LIN {X -0.197,Y -544.283,Z 869.058,A 0.000,B 0.000,C 90.000,E1 46.458} C_DIS
LIN {X -0.178,Y -541.892,Z 869.055,A 0.000,B 0.000,C 90.000,E1 45.891} C_DIS
LIN {X 0.010,Y -538.422,Z 869.051,A 0.000,B 0.000,C 90.000,E1 45.162} C_DIS
LIN {X -0.016,Y -535.445,Z 869.048,A 0.000,B 0.000,C 90.000,E1 44.595} C_DIS
LIN {X -0.036,Y -532.256,Z 869.045,A 0.000,B 0.000,C 90.000,E1 44.028} C_DIS
LIN {X 0.058,Y -527.783,Z 869.041,A 0.000,B 0.000,C 90.000,E1 43.299} C_DIS
LIN {X -0.050,Y -524.016,Z 869.037,A 0.000,B 0.000,C 90.000,E1 42.732} C_DIS
LIN {X -0.151,Y -519.980,Z 869.034,A 0.000,B 0.000,C 90.000,E1 42.162} C_DIS
LIN {X 0.073,Y -515.730,Z 869.031,A 0.000,B 0.000,C 90.000,E1 41.553} C_DIS
LIN {X -0.182,Y -512.399,Z 869.029,A 0.000,B 0.000,C 90.000,E1 41.148} C_DIS
LIN {X -0.002,Y -503.778,Z 869.023,A 0.000,B 0.000,C 90.000,E1 40.092} C_DIS
LIN {X 0.166,Y -498.386,Z 869.020,A 0.000,B 0.000,C 90.000,E1 39.483} C_DIS
LIN {X -0.295,Y -491.480,Z 869.016,A 0.000,B 0.000,C 90.000,E1 38.830} C_DIS
LIN {X -0.121,Y -485.726,Z 869.013,A 0.000,B 0.000,C 90.000,E1 38.257} C_DIS
LIN {X 0.040,Y -478.343,Z 869.009,A 0.000,B 0.000,C 90.000,E1 37.569} C_DIS
LIN {X 0.098,Y -467.773,Z 869.004,A 0.000,B 0.000,C 90.000,E1 36.664} C_DIS
LIN {X -0.016,Y -456.899,Z 868.999,A 0.000,B 0.000,C 90.000,E1 35.804} C_DIS
LIN {X 0.026,Y -444.305,Z 868.994,A 0.000,B 0.000,C 90.000,E1 34.818} C_DIS
LIN {X -0.079,Y -422.825,Z 868.984,A 0.000,B 0.000,C 90.000,E1 33.086} C_DIS
LIN {X -0.077,Y -409.157,Z 868.977,A 0.000,B 0.000,C 90.000,E1 31.878} C_DIS
LIN {X 0.140,Y -401.842,Z 868.973,A 0.000,B 0.000,C 90.000,E1 31.131} C_DIS
LIN {X -0.162,Y -396.543,Z 868.970,A 0.000,B 0.000,C 90.000,E1 30.541} C_DIS
LIN {X -0.062,Y -394.558,Z 868.968,A 0.000,B 0.000,C 90.000,E1 30.256} C_DIS
LIN {X -0.054,Y -393.500,Z 868.967,A 0.000,B 0.000,C 90.000,E1 30.079} C_DIS
LIN {X 0.085,Y -391.376,Z 868.965,A 0.000,B 0.000,C 90.000,E1 29.617} C_DIS
LIN {X 0.058,Y -390.008,Z 868.961,A 0.000,B 0.000,C 90.000,E1 28.999} C_DIS
LIN {X -0.092,Y -389.501,Z 868.958,A 0.000,B 0.000,C 90.000,E1 28.487} C_DIS
LIN {X 0.127,Y -389.595,Z 868.952,A 0.000,B 0.000,C 90.000,E1 27.385} C_DIS
LIN {X -0.188,Y -392.234,Z 868.931,A 0.000,B 0.000,C 90.000,E1 23.515} C_DIS
LIN {X -0.027,Y -395.272,Z 868.913,A 0.000,B 0.000,C 90.000,E1 20.301} C_DIS
LIN {X 0.136,Y -398.327,Z 868.897,A 0.000,B 0.000,C 90.000,E1 17.457} C_DIS
LIN {X -0.006,Y -400.906,Z 868.885,A 0.000,B 0.000,C 90.000,E1 15.371} C_DIS
LIN {X -0.105,Y -405.159,Z 868.868,A 0.000,B 0.000,C 90.000,E1 12.243} C_DIS
LIN {X 0.056,Y -408.867,Z 868.854,A 0.000,B 0.000,C 90.000,E1 9.792} C_DIS
LIN {X -0.142,Y -414.004,Z 868.837,A 0.000,B 0.000,C 90.000,E1 6.720} C_DIS
LIN {X 0.028,Y -417.746,Z 868.826,A 0.000,B 0.000,C 90.000,E1 4.645} C_DIS
LIN {X -0.123,Y -423.210,Z 868.811,A 0.000,B 0.000,C 90.000,E1 1.949} C_DIS
LIN {X -0.136,Y -429.645,Z 868.795,A 0.000,B 0.000,C 90.000,E1 359.141} C_DIS
LIN {X 0.105,Y -436.193,Z 868.780,A 0.000,B 0.000,C 90.000,E1 356.445} C_DIS
LIN {X 0.117,Y -439.553,Z 868.773,A 0.000,B 0.000,C 90.000,E1 355.122} C_DIS
LIN {X -0.022,Y -442.286,Z 868.768,A 0.000,B 0.000,C 90.000,E1 354.318} C_DIS
LIN {X 0.133,Y -443.631,Z 868.767,A 0.000,B 0.000,C 90.000,E1 353.970} C_DIS
LIN {X 0.004,Y -445.225,Z 868.765,A 0.000,B 0.000,C 90.000,E1 353.685} C_DIS
LIN {X -0.182,Y -446.287,Z 868.764,A 0.000,B 0.000,C 90.000,E1 353.571} C_DIS
LIN {X 0.011,Y -448.820,Z 868.763,A 0.000,B 0.000,C 90.000,E1 353.280} C_DIS
LIN {X 0.203,Y -450.563,Z 868.762,A 0.000,B 0.000,C 90.000,E1 353.109} C_DIS
LIN {X -0.101,Y -457.050,Z 868.760,A 0.000,B 0.000,C 90.000,E1 352.761} C_DIS
LIN {X 0.066,Y -466.908,Z 868.757,A 0.000,B 0.000,C 90.000,E1 352.299} C_DIS
LIN {X -0.142,Y -476.793,Z 868.755,A 0.000,B 0.000,C 90.000,E1 351.837} C_DIS
LIN {X 0.080,Y -484.903,Z 868.752,A 0.000,B 0.000,C 90.000,E1 351.376} C_DIS
LIN {X -0.128,Y -491.410,Z 868.750,A 0.000,B 0.000,C 90.000,E1 351.027} C_DIS
LIN {X 0.259,Y -499.429,Z 868.747,A 0.000,B 0.000,C 90.000,E1 350.500} C_DIS
LIN {X 0.071,Y -510.569,Z 868.743,A 0.000,B 0.000,C 90.000,E1 349.803} C_DIS
LIN {X 0.001,Y -518.351,Z 868.741,A 0.000,B 0.000,C 90.000,E1 349.285} C_DIS
LIN {X -0.143,Y -525.997,Z 868.737,A 0.000,B 0.000,C 90.000,E1 348.757} C_DIS
LIN {X 0.082,Y -531.968,Z 868.735,A 0.000,B 0.000,C 90.000,E1 348.285} C_DIS
LIN {X 0.031,Y -540.629,Z 868.731,A 0.000,B 0.000,C 90.000,E1 347.589} C_DIS
LIN {X 0.017,Y -544.852,Z 868.729,A 0.000,B 0.000,C 90.000,E1 347.229} C_DIS
LIN {X 0.273,Y -550.376,Z 868.726,A 0.000,B 0.000,C 90.000,E1 346.700} C_DIS
LIN {X 0.133,Y -558.287,Z 868.722,A 0.000,B 0.000,C 90.000,E1 345.936} C_DIS
LIN {X -0.219,Y -562.102,Z 868.720,A 0.000,B 0.000,C 90.000,E1 345.574} C_DIS
LIN {X 0.194,Y -567.029,Z 868.717,A 0.000,B 0.000,C 90.000,E1 344.991} C_DIS
LIN {X 0.145,Y -571.768,Z 868.714,A 0.000,B 0.000,C 90.000,E1 344.448} C_DIS
LIN {X 0.065,Y -579.478,Z 868.708,A 0.000,B 0.000,C 90.000,E1 343.504} C_DIS
LIN {X 0.015,Y -584.516,Z 868.705,A 0.000,B 0.000,C 90.000,E1 342.834} C_DIS
LIN {X -0.166,Y -589.155,Z 868.701,A 0.000,B 0.000,C 90.000,E1 342.181} C_DIS
LIN {X 0.125,Y -595.226,Z 868.696,A 0.000,B 0.000,C 90.000,E1 341.221} C_DIS
LIN {X -0.081,Y -600.727,Z 868.691,A 0.000,B 0.000,C 90.000,E1 340.315} C_DIS
LIN {X -0.086,Y -607.372,Z 868.684,A 0.000,B 0.000,C 90.000,E1 339.135} C_DIS
LIN {X 0.329,Y -615.013,Z 868.676,A 0.000,B 0.000,C 90.000,E1 337.667} C_DIS
LIN {X 0.004,Y -619.578,Z 868.671,A 0.000,B 0.000,C 90.000,E1 336.794} C_DIS
LIN {X -0.271,Y -622.717,Z 868.668,A 0.000,B 0.000,C 90.000,E1 336.177} C_DIS
LIN {X 0.305,Y -626.226,Z 868.663,A 0.000,B 0.000,C 90.000,E1 335.357} C_DIS
LIN {X 0.350,Y -629.645,Z 868.659,A 0.000,B 0.000,C 90.000,E1 334.588} C_DIS
LIN {X -0.342,Y -634.773,Z 868.652,A 0.000,B 0.000,C 90.000,E1 333.384} C_DIS
LIN {X -0.161,Y -638.648,Z 868.646,A 0.000,B 0.000,C 90.000,E1 332.359} C_DIS
LIN {X 0.374,Y -642.199,Z 868.641,A 0.000,B 0.000,C 90.000,E1 331.307} C_DIS
LIN {X 0.087,Y -645.573,Z 868.635,A 0.000,B 0.000,C 90.000,E1 330.333} C_DIS
LIN {X 0.161,Y -648.796,Z 868.630,A 0.000,B 0.000,C 90.000,E1 329.331} C_DIS
LIN {X -0.185,Y -652.505,Z 868.623,A 0.000,B 0.000,C 90.000,E1 328.122} C_DIS
LIN {X -0.114,Y -654.551,Z 868.619,A 0.000,B 0.000,C 90.000,E1 327.375} C_DIS
LIN {X 0.069,Y -657.145,Z 868.613,A 0.000,B 0.000,C 90.000,E1 326.373} C_DIS
LIN {X -0.342,Y -659.954,Z 868.606,A 0.000,B 0.000,C 90.000,E1 325.182} C_DIS
LIN {X 0.218,Y -662.343,Z 868.600,A 0.000,B 0.000,C 90.000,E1 323.909} C_DIS
LIN {X -0.208,Y -664.036,Z 868.594,A 0.000,B 0.000,C 90.000,E1 322.970} C_DIS
LIN {X -0.110,Y -665.856,Z 868.587,A 0.000,B 0.000,C 90.000,E1 321.743} C_DIS
LIN {X 0.008,Y -667.448,Z 868.581,A 0.000,B 0.000,C 90.000,E1 320.517} C_DIS
LIN {X 0.061,Y -668.583,Z 868.575,A 0.000,B 0.000,C 90.000,E1 319.542} C_DIS
LIN {X 0.128,Y -669.707,Z 868.570,A 0.000,B 0.000,C 90.000,E1 318.566} C_DIS
LIN {X 0.260,Y -672.002,Z 868.558,A 0.000,B 0.000,C 90.000,E1 316.377} C_DIS
LIN {X 0.357,Y -673.553,Z 868.551,A 0.000,B 0.000,C 90.000,E1 315.162} C_DIS
LIN {X -0.053,Y -674.252,Z 868.547,A 0.000,B 0.000,C 90.000,E1 314.474} C_DIS
LIN {X -0.029,Y -674.367,Z 868.546,A 0.000,B 0.000,C 90.000,E1 314.231} C_DIS
LIN {X 0.122,Y -675.592,Z 868.539,A 0.000,B 0.000,C 90.000,E1 313.014} C_DIS
LIN {X -0.163,Y -677.036,Z 868.531,A 0.000,B 0.000,C 90.000,E1 311.595} C_DIS
LIN {X 0.044,Y -678.135,Z 868.524,A 0.000,B 0.000,C 90.000,E1 310.378} C_DIS
LIN {X -0.143,Y -679.336,Z 868.516,A 0.000,B 0.000,C 90.000,E1 308.955} C_DIS
LIN {X 0.194,Y -680.311,Z 868.510,A 0.000,B 0.000,C 90.000,E1 307.729} C_DIS
LIN {X -0.402,Y -681.261,Z 868.503,A 0.000,B 0.000,C 90.000,E1 306.583} C_DIS
LIN {X -0.035,Y -682.140,Z 868.496,A 0.000,B 0.000,C 90.000,E1 305.358} C_DIS
LIN {X 0.124,Y -683.066,Z 868.489,A 0.000,B 0.000,C 90.000,E1 303.913} C_DIS
LIN {X -0.256,Y -684.589,Z 868.477,A 0.000,B 0.000,C 90.000,E1 301.799} C_DIS
LIN {X -0.203,Y -685.887,Z 868.467,A 0.000,B 0.000,C 90.000,E1 300.129} C_DIS
LIN {X -0.171,Y -688.321,Z 868.453,A 0.000,B 0.000,C 90.000,E1 297.513} C_DIS
LIN {X -0.325,Y -689.775,Z 868.445,A 0.000,B 0.000,C 90.000,E1 296.104} C_DIS
LIN {X -0.303,Y -690.807,Z 868.440,A 0.000,B 0.000,C 90.000,E1 295.155} C_DIS
LIN {X -0.032,Y -691.777,Z 868.433,A 0.000,B 0.000,C 90.000,E1 293.951} C_DIS
LIN {X 0.168,Y -691.864,Z 868.430,A 0.000,B 0.000,C 90.000,E1 293.462} C_DIS
LIN {X -0.230,Y -691.797,Z 868.429,A 0.000,B 0.000,C 90.000,E1 293.259} C_DIS
LIN {X -0.028,Y -691.076,Z 868.427,A 0.000,B 0.000,C 90.000,E1 292.770} C_DIS
LIN {X 0.205,Y -690.377,Z 868.425,A 0.000,B 0.000,C 90.000,E1 292.514} C_DIS
LIN {X 0.286,Y -688.409,Z 868.423,A 0.000,B 0.000,C 90.000,E1 292.153} C_DIS
LIN {X -0.129,Y -686.936,Z 868.422,A 0.000,B 0.000,C 90.000,E1 291.950} C_DIS
LIN {X -0.275,Y -685.791,Z 868.421,A 0.000,B 0.000,C 90.000,E1 291.844} C_DIS
LIN {X -0.168,Y -684.078,Z 868.421,A 0.000,B 0.000,C 90.000,E1 291.716} C_DIS
LIN {X 0.160,Y -680.344,Z 868.419,A 0.000,B 0.000,C 90.000,E1 291.482} C_DIS
LIN {X -0.041,Y -676.937,Z 868.419,A 0.000,B 0.000,C 90.000,E1 291.334} C_DIS
LIN {X -0.144,Y -670.811,Z 868.417,A 0.000,B 0.000,C 90.000,E1 291.153} C_DIS
LIN {X -0.224,Y -658.370,Z 868.416,A 0.000,B 0.000,C 90.000,E1 290.844} C_DIS
LIN {X 0.181,Y -654.807,Z 868.415,A 0.000,B 0.000,C 90.000,E1 290.684} C_DIS
LIN {X -0.260,Y -652.134,Z 868.414,A 0.000,B 0.000,C 90.000,E1 290.610} C_DIS
LIN {X -0.212,Y -650.429,Z 868.414,A 0.000,B 0.000,C 90.000,E1 290.482} C_DIS
LIN {X 0.072,Y -649.078,Z 868.413,A 0.000,B 0.000,C 90.000,E1 290.355} C_DIS
LIN {X 0.034,Y -649.065,Z 868.413,A 0.000,B 0.000,C 90.000,E1 290.355} C_DIS
LIN {X -0.066,Y -648.618,Z 868.412,A 0.000,B 0.000,C 90.000,E1 290.248} C_DIS
LIN {X -0.110,Y -648.618,Z 868.412,A 0.000,B 0.000,C 90.000,E1 290.248} C_DIS
LIN {X -0.132,Y -649.438,Z 868.410,A 0.000,B 0.000,C 90.000,E1 289.885} C_DIS
LIN {X -0.167,Y -652.192,Z 868.407,A 0.000,B 0.000,C 90.000,E1 289.268} C_DIS
LIN {X 0.241,Y -658.845,Z 868.400,A 0.000,B 0.000,C 90.000,E1 288.000} C_DIS
LIN {X 0.117,Y -662.385,Z 868.396,A 0.000,B 0.000,C 90.000,E1 287.275} C_DIS
LIN {X 0.021,Y -665.410,Z 868.392,A 0.000,B 0.000,C 90.000,E1 286.551} C_DIS
LIN {X -0.153,Y -667.161,Z 868.389,A 0.000,B 0.000,C 90.000,E1 286.079} C_DIS
LIN {X -0.389,Y -669.411,Z 868.385,A 0.000,B 0.000,C 90.000,E1 285.371} C_DIS
LIN {X 0.288,Y -670.650,Z 868.383,A 0.000,B 0.000,C 90.000,E1 284.828} C_DIS
LIN {X 0.023,Y -672.437,Z 868.377,A 0.000,B 0.000,C 90.000,E1 283.883} C_DIS
LIN {X -0.040,Y -672.850,Z 868.376,A 0.000,B 0.000,C 90.000,E1 283.647} C_DIS
LIN {X 0.377,Y -673.880,Z 868.370,A 0.000,B 0.000,C 90.000,E1 282.647} C_DIS
LIN {X 0.062,Y -674.337,Z 868.366,A 0.000,B 0.000,C 90.000,E1 281.951} C_DIS
LIN {X -0.109,Y -674.352,Z 868.362,A 0.000,B 0.000,C 90.000,E1 281.243} C_DIS
LIN {X -0.354,Y -674.152,Z 868.360,A 0.000,B 0.000,C 90.000,E1 280.782} C_DIS
LIN {X 0.189,Y -673.702,Z 868.357,A 0.000,B 0.000,C 90.000,E1 280.254} C_DIS
LIN {X -0.052,Y -672.960,Z 868.354,A 0.000,B 0.000,C 90.000,E1 279.792} C_DIS
LIN {X -0.184,Y -671.934,Z 868.352,A 0.000,B 0.000,C 90.000,E1 279.321} C_DIS
LIN {X 0.230,Y -670.570,Z 868.349,A 0.000,B 0.000,C 90.000,E1 278.803} C_DIS
LIN {X -0.024,Y -668.909,Z 868.346,A 0.000,B 0.000,C 90.000,E1 278.341} C_DIS
LIN {X -0.107,Y -668.021,Z 868.345,A 0.000,B 0.000,C 90.000,E1 278.106} C_DIS
LIN {X 0.286,Y -665.917,Z 868.342,A 0.000,B 0.000,C 90.000,E1 277.587} C_DIS
LIN {X -0.006,Y -662.895,Z 868.339,A 0.000,B 0.000,C 90.000,E1 277.004} C_DIS
LIN {X 0.346,Y -660.140,Z 868.336,A 0.000,B 0.000,C 90.000,E1 276.486} C_DIS
LIN {X -0.077,Y -656.035,Z 868.333,A 0.000,B 0.000,C 90.000,E1 275.910} C_DIS
LIN {X 0.227,Y -652.239,Z 868.330,A 0.000,B 0.000,C 90.000,E1 275.391} C_DIS
LIN {X -0.258,Y -646.569,Z 868.327,A 0.000,B 0.000,C 90.000,E1 274.816} C_DIS
LIN {X 0.058,Y -641.662,Z 868.324,A 0.000,B 0.000,C 90.000,E1 274.302} C_DIS
LIN {X -0.051,Y -636.315,Z 868.321,A 0.000,B 0.000,C 90.000,E1 273.841} C_DIS
LIN {X 0.009,Y -630.719,Z 868.319,A 0.000,B 0.000,C 90.000,E1 273.383} C_DIS
LIN {X -0.187,Y -624.915,Z 868.317,A 0.000,B 0.000,C 90.000,E1 272.980} C_DIS
LIN {X 0.116,Y -617.299,Z 868.314,A 0.000,B 0.000,C 90.000,E1 272.465} C_DIS
LIN {X -0.126,Y -610.630,Z 868.312,A 0.000,B 0.000,C 90.000,E1 272.121} C_DIS
LIN {X -0.022,Y -603.828,Z 868.310,A 0.000,B 0.000,C 90.000,E1 271.776} C_DIS
LIN {X -0.152,Y -596.472,Z 868.308,A 0.000,B 0.000,C 90.000,E1 271.489} C_DIS
LIN {X 0.194,Y -591.084,Z 868.307,A 0.000,B 0.000,C 90.000,E1 271.260} C_DIS
LIN {X 0.273,Y -583.480,Z 868.306,A 0.000,B 0.000,C 90.000,E1 271.031} C_DIS
LIN {X 0.109,Y -577.567,Z 868.305,A 0.000,B 0.000,C 90.000,E1 270.917} C_DIS
LIN {X 0.132,Y -571.301,Z 868.305,A 0.000,B 0.000,C 90.000,E1 270.802} C_DIS
LIN {X -0.095,Y -564.097,Z 868.304,A 0.000,B 0.000,C 90.000,E1 270.745} C_DIS
LIN {X -0.109,Y -552.668,Z 868.304,A 0.000,B 0.000,C 90.000,E1 270.688} C_DIS
LIN {X 0.187,Y -549.596,Z 868.303,A 0.000,B 0.000,C 90.000,E1 270.573} C_DIS
LIN {X 0.157,Y -549.518,Z 868.303,A 0.000,B 0.000,C 90.000,E1 270.573} C_DIS
LIN {X -0.177,Y -547.454,Z 868.302,A 0.000,B 0.000,C 90.000,E1 270.344} C_DIS
LIN {X 0.153,Y -546.964,Z 868.301,A 0.000,B 0.000,C 90.000,E1 270.172} C_DIS
LIN {X -0.068,Y -545.980,Z 868.298,A 0.000,B 0.000,C 90.000,E1 269.714} C_DIS
LIN {X 0.180,Y -544.198,Z 868.289,A 0.000,B 0.000,C 90.000,E1 267.993} C_DIS
LIN {X -0.065,Y -542.539,Z 868.276,A 0.000,B 0.000,C 90.000,E1 265.755} C_DIS
LIN {X 0.132,Y -541.407,Z 868.267,A 0.000,B 0.000,C 90.000,E1 264.033} C_DIS
LIN {X -0.193,Y -540.299,Z 868.259,A 0.000,B 0.000,C 90.000,E1 262.648} C_DIS
LIN {X 0.143,Y -538.737,Z 868.250,A 0.000,B 0.000,C 90.000,E1 260.905} C_DIS
LIN {X -0.077,Y -537.063,Z 868.240,A 0.000,B 0.000,C 90.000,E1 259.218} C_DIS
LIN {X 0.172,Y -535.823,Z 868.234,A 0.000,B 0.000,C 90.000,E1 258.049} C_DIS
LIN {X -0.123,Y -534.523,Z 868.227,A 0.000,B 0.000,C 90.000,E1 256.937} C_DIS
LIN {X 0.247,Y -532.762,Z 868.219,A 0.000,B 0.000,C 90.000,E1 255.463} C_DIS
LIN {X 0.062,Y -531.010,Z 868.211,A 0.000,B 0.000,C 90.000,E1 254.047} C_DIS
LIN {X 0.159,Y -528.989,Z 868.202,A 0.000,B 0.000,C 90.000,E1 252.308} C_DIS
LIN {X 0.200,Y -527.579,Z 868.195,A 0.000,B 0.000,C 90.000,E1 251.148} C_DIS
LIN {X 0.221,Y -525.670,Z 868.187,A 0.000,B 0.000,C 90.000,E1 249.699} C_DIS
LIN {X -0.106,Y -523.660,Z 868.179,A 0.000,B 0.000,C 90.000,E1 248.284} C_DIS
LIN {X 0.212,Y -521.516,Z 868.171,A 0.000,B 0.000,C 90.000,E1 246.794} C_DIS
LIN {X -0.135,Y -519.738,Z 868.165,A 0.000,B 0.000,C 90.000,E1 245.665} C_DIS
LIN {X -0.018,Y -517.017,Z 868.155,A 0.000,B 0.000,C 90.000,E1 243.896} C_DIS
LIN {X -0.196,Y -514.052,Z 868.145,A 0.000,B 0.000,C 90.000,E1 242.153} C_DIS
LIN {X -0.106,Y -510.431,Z 868.134,A 0.000,B 0.000,C 90.000,E1 240.078} C_DIS
LIN {X 0.099,Y -508.251,Z 868.127,A 0.000,B 0.000,C 90.000,E1 238.869} C_DIS
LIN {X -0.155,Y -506.003,Z 868.121,A 0.000,B 0.000,C 90.000,E1 237.709} C_DIS
LIN {X -0.127,Y -503.122,Z 868.112,A 0.000,B 0.000,C 90.000,E1 236.215} C_DIS
LIN {X -0.054,Y -501.273,Z 868.107,A 0.000,B 0.000,C 90.000,E1 235.308} C_DIS
LIN {X -0.125,Y -498.475,Z 868.101,A 0.000,B 0.000,C 90.000,E1 234.116} C_DIS
LIN {X -0.077,Y -494.841,Z 868.092,A 0.000,B 0.000,C 90.000,E1 232.603} C_DIS
LIN {X -0.094,Y -489.786,Z 868.080,A 0.000,B 0.000,C 90.000,E1 230.481} C_DIS
LIN {X 0.089,Y -486.326,Z 868.072,A 0.000,B 0.000,C 90.000,E1 228.933} C_DIS
LIN {X 0.219,Y -480.908,Z 868.058,A 0.000,B 0.000,C 90.000,E1 226.458} C_DIS
LIN {X -0.063,Y -476.891,Z 868.048,A 0.000,B 0.000,C 90.000,E1 224.636} C_DIS
LIN {X -0.174,Y -475.534,Z 868.045,A 0.000,B 0.000,C 90.000,E1 224.028} C_DIS
LIN {X -0.131,Y -470.766,Z 868.032,A 0.000,B 0.000,C 90.000,E1 221.838} C_DIS
LIN {X 0.060,Y -466.660,Z 868.022,A 0.000,B 0.000,C 90.000,E1 219.930} C_DIS
LIN {X -0.041,Y -461.947,Z 868.010,A 0.000,B 0.000,C 90.000,E1 217.729} C_DIS
LIN {X -0.026,Y -458.644,Z 868.001,A 0.000,B 0.000,C 90.000,E1 216.137} C_DIS
LIN {X 0.125,Y -454.560,Z 867.990,A 0.000,B 0.000,C 90.000,E1 214.199} C_DIS
LIN {X -0.272,Y -449.041,Z 867.976,A 0.000,B 0.000,C 90.000,E1 211.671} C_DIS
LIN {X 0.107,Y -445.582,Z 867.967,A 0.000,B 0.000,C 90.000,E1 210.001} C_DIS
LIN {X 0.033,Y -441.445,Z 867.956,A 0.000,B 0.000,C 90.000,E1 208.052} C_DIS
LIN {X -0.113,Y -436.579,Z 867.943,A 0.000,B 0.000,C 90.000,E1 205.771} C_DIS
LIN {X 0.001,Y -432.360,Z 867.932,A 0.000,B 0.000,C 90.000,E1 203.770} C_DIS
LIN {X 0.048,Y -429.001,Z 867.923,A 0.000,B 0.000,C 90.000,E1 202.099} C_DIS
LIN {X 0.029,Y -425.565,Z 867.914,A 0.000,B 0.000,C 90.000,E1 200.429} C_DIS
LIN {X -0.034,Y -421.585,Z 867.902,A 0.000,B 0.000,C 90.000,E1 198.417} C_DIS
LIN {X 0.137,Y -418.994,Z 867.895,A 0.000,B 0.000,C 90.000,E1 197.040} C_DIS
LIN {X -0.136,Y -416.226,Z 867.887,A 0.000,B 0.000,C 90.000,E1 195.717} C_DIS
LIN {X -0.130,Y -412.786,Z 867.878,A 0.000,B 0.000,C 90.000,E1 194.008} C_DIS
LIN {X -0.056,Y -408.051,Z 867.864,A 0.000,B 0.000,C 90.000,E1 191.591} C_DIS
LIN {X 0.013,Y -405.331,Z 867.857,A 0.000,B 0.000,C 90.000,E1 190.197} C_DIS
LIN {X 0.042,Y -401.878,Z 867.847,A 0.000,B 0.000,C 90.000,E1 188.454} C_DIS
LIN {X 0.085,Y -394.628,Z 867.826,A 0.000,B 0.000,C 90.000,E1 184.588} C_DIS
LIN {X 0.054,Y -388.590,Z 867.804,A 0.000,B 0.000,C 90.000,E1 180.688} C_DIS
LIN {X -0.022,Y -386.099,Z 867.794,A 0.000,B 0.000,C 90.000,E1 178.912} C_DIS
LIN {X -0.143,Y -383.551,Z 867.784,A 0.000,B 0.000,C 90.000,E1 177.135} C_DIS
LIN {X 0.081,Y -380.945,Z 867.774,A 0.000,B 0.000,C 90.000,E1 175.298} C_DIS
LIN {X -0.126,Y -376.593,Z 867.756,A 0.000,B 0.000,C 90.000,E1 172.064} C_DIS
LIN {X 0.117,Y -373.744,Z 867.740,A 0.000,B 0.000,C 90.000,E1 169.106} C_DIS
LIN {X -0.037,Y -373.143,Z 867.729,A 0.000,B 0.000,C 90.000,E1 167.297} C_DIS
LIN {X -0.200,Y -373.065,Z 867.725,A 0.000,B 0.000,C 90.000,E1 166.589} C_DIS
LIN {X -0.036,Y -373.482,Z 867.719,A 0.000,B 0.000,C 90.000,E1 165.463} C_DIS
LIN {X -0.198,Y -374.026,Z 867.715,A 0.000,B 0.000,C 90.000,E1 164.755} C_DIS
LIN {X 0.106,Y -375.078,Z 867.711,A 0.000,B 0.000,C 90.000,E1 163.976} C_DIS
LIN {X -0.045,Y -376.748,Z 867.707,A 0.000,B 0.000,C 90.000,E1 163.268} C_DIS
LIN {X -0.071,Y -378.591,Z 867.704,A 0.000,B 0.000,C 90.000,E1 162.725} C_DIS
LIN {X -0.084,Y -382.638,Z 867.700,A 0.000,B 0.000,C 90.000,E1 162.000} C_DIS
LIN {X 0.046,Y -388.965,Z 867.696,A 0.000,B 0.000,C 90.000,E1 161.329} C_DIS
LIN {X -0.154,Y -392.565,Z 867.695,A 0.000,B 0.000,C 90.000,E1 161.094} C_DIS
LIN {X 0.057,Y -396.273,Z 867.694,A 0.000,B 0.000,C 90.000,E1 160.859} C_DIS
LIN {X -0.075,Y -407.283,Z 867.691,A 0.000,B 0.000,C 90.000,E1 160.369} C_DIS
LIN {X 0.119,Y -412.241,Z 867.690,A 0.000,B 0.000,C 90.000,E1 160.115} C_DIS
LIN {X -0.076,Y -422.368,Z 867.687,A 0.000,B 0.000,C 90.000,E1 159.625} C_DIS
LIN {X -0.111,Y -428.851,Z 867.685,A 0.000,B 0.000,C 90.000,E1 159.263} C_DIS
LIN {X 0.158,Y -432.122,Z 867.684,A 0.000,B 0.000,C 90.000,E1 159.028} C_DIS
LIN {X 0.185,Y -438.265,Z 867.681,A 0.000,B 0.000,C 90.000,E1 158.592} C_DIS
LIN {X -0.013,Y -444.685,Z 867.679,A 0.000,B 0.000,C 90.000,E1 158.156} C_DIS
LIN {X -0.023,Y -452.335,Z 867.675,A 0.000,B 0.000,C 90.000,E1 157.539} C_DIS
LIN {X 0.079,Y -459.657,Z 867.672,A 0.000,B 0.000,C 90.000,E1 156.869} C_DIS
LIN {X -0.130,Y -464.014,Z 867.669,A 0.000,B 0.000,C 90.000,E1 156.485} C_DIS
LIN {X 0.116,Y -475.059,Z 867.663,A 0.000,B 0.000,C 90.000,E1 155.305} C_DIS
LIN {X 0.141,Y -480.397,Z 867.660,A 0.000,B 0.000,C 90.000,E1 154.717} C_DIS
LIN {X 0.080,Y -486.875,Z 867.656,A 0.000,B 0.000,C 90.000,E1 153.973} C_DIS
LIN {X 0.126,Y -492.956,Z 867.651,A 0.000,B 0.000,C 90.000,E1 153.204} C_DIS
LIN {X -0.267,Y -504.284,Z 867.643,A 0.000,B 0.000,C 90.000,E1 151.769} C_DIS
LIN {X -0.152,Y -507.524,Z 867.641,A 0.000,B 0.000,C 90.000,E1 151.307} C_DIS
LIN {X -0.031,Y -514.896,Z 867.635,A 0.000,B 0.000,C 90.000,E1 150.255} C_DIS
LIN {X 0.149,Y -517.786,Z 867.632,A 0.000,B 0.000,C 90.000,E1 149.793} C_DIS
LIN {X -0.193,Y -519.767,Z 867.631,A 0.000,B 0.000,C 90.000,E1 149.537} C_DIS
LIN {X 0.016,Y -522.734,Z 867.628,A 0.000,B 0.000,C 90.000,E1 149.076} C_DIS
LIN {X 0.035,Y -528.210,Z 867.623,A 0.000,B 0.000,C 90.000,E1 148.201} C_DIS
LIN {X 0.114,Y -533.412,Z 867.619,A 0.000,B 0.000,C 90.000,E1 147.327} C_DIS
LIN {X -0.343,Y -540.754,Z 867.611,A 0.000,B 0.000,C 90.000,E1 146.087} C_DIS
LIN {X 0.172,Y -545.299,Z 867.607,A 0.000,B 0.000,C 90.000,E1 145.182} C_DIS
LIN {X 0.218,Y -551.991,Z 867.600,A 0.000,B 0.000,C 90.000,E1 143.909} C_DIS
LIN {X 0.087,Y -556.383,Z 867.595,A 0.000,B 0.000,C 90.000,E1 143.084} C_DIS
LIN {X 0.076,Y -563.544,Z 867.587,A 0.000,B 0.000,C 90.000,E1 141.698} C_DIS
LIN {X -0.245,Y -570.774,Z 867.580,A 0.000,B 0.000,C 90.000,E1 140.356} C_DIS
LIN {X 0.011,Y -573.577,Z 867.577,A 0.000,B 0.000,C 90.000,E1 139.784} C_DIS
LIN {X -0.033,Y -579.444,Z 867.570,A 0.000,B 0.000,C 90.000,E1 138.566} C_DIS
LIN {X 0.119,Y -591.123,Z 867.556,A 0.000,B 0.000,C 90.000,E1 136.134} C_DIS
LIN {X -0.089,Y -596.837,Z 867.550,A 0.000,B 0.000,C 90.000,E1 134.960} C_DIS
LIN {X 0.018,Y -603.677,Z 867.542,A 0.000,B 0.000,C 90.000,E1 133.500} C_DIS
LIN {X -0.111,Y -609.461,Z 867.534,A 0.000,B 0.000,C 90.000,E1 132.204} C_DIS
LIN {X 0.066,Y -614.106,Z 867.529,A 0.000,B 0.000,C 90.000,E1 131.148} C_DIS
LIN {X 0.143,Y -619.325,Z 867.521,A 0.000,B 0.000,C 90.000,E1 129.850} C_DIS
LIN {X -0.096,Y -624.303,Z 867.514,A 0.000,B 0.000,C 90.000,E1 128.588} C_DIS
LIN {X -0.304,Y -626.304,Z 867.512,A 0.000,B 0.000,C 90.000,E1 128.096} C_DIS
LIN {X 0.275,Y -633.863,Z 867.500,A 0.000,B 0.000,C 90.000,E1 126.011} C_DIS
LIN {X 0.010,Y -637.284,Z 867.495,A 0.000,B 0.000,C 90.000,E1 125.025} C_DIS
LIN {X 0.316,Y -640.438,Z 867.489,A 0.000,B 0.000,C 90.000,E1 123.992} C_DIS
LIN {X -0.271,Y -642.596,Z 867.485,A 0.000,B 0.000,C 90.000,E1 123.293} C_DIS
LIN {X 0.183,Y -644.109,Z 867.482,A 0.000,B 0.000,C 90.000,E1 122.752} C_DIS
LIN {X 0.167,Y -645.929,Z 867.478,A 0.000,B 0.000,C 90.000,E1 122.005} C_DIS
LIN {X -0.243,Y -646.909,Z 867.475,A 0.000,B 0.000,C 90.000,E1 121.544} C_DIS
LIN {X 0.245,Y -648.089,Z 867.472,A 0.000,B 0.000,C 90.000,E1 121.003} C_DIS
LIN {X 0.265,Y -649.593,Z 867.468,A 0.000,B 0.000,C 90.000,E1 120.256} C_DIS
LIN {X 0.163,Y -651.642,Z 867.461,A 0.000,B 0.000,C 90.000,E1 119.027} C_DIS
LIN {X -0.209,Y -652.474,Z 867.459,A 0.000,B 0.000,C 90.000,E1 118.565} C_DIS
LIN {X 0.307,Y -653.102,Z 867.456,A 0.000,B 0.000,C 90.000,E1 118.025} C_DIS
LIN {X 0.045,Y -654.272,Z 867.452,A 0.000,B 0.000,C 90.000,E1 117.308} C_DIS
LIN {X 0.198,Y -655.731,Z 867.446,A 0.000,B 0.000,C 90.000,E1 116.309} C_DIS
LIN {X -0.159,Y -656.272,Z 867.444,A 0.000,B 0.000,C 90.000,E1 115.848} C_DIS
LIN {X 0.152,Y -657.228,Z 867.437,A 0.000,B 0.000,C 90.000,E1 114.591} C_DIS
LIN {X -0.208,Y -657.292,Z 867.434,A 0.000,B 0.000,C 90.000,E1 114.131} C_DIS
LIN {X -0.239,Y -657.057,Z 867.431,A 0.000,B 0.000,C 90.000,E1 113.643} C_DIS
LIN {X -0.122,Y -656.742,Z 867.430,A 0.000,B 0.000,C 90.000,E1 113.387} C_DIS
LIN {X -0.150,Y -654.997,Z 867.427,A 0.000,B 0.000,C 90.000,E1 112.898} C_DIS
LIN {X -0.095,Y -654.441,Z 867.427,A 0.000,B 0.000,C 90.000,E1 112.770} C_DIS
LIN {X 0.012,Y -652.332,Z 867.425,A 0.000,B 0.000,C 90.000,E1 112.514} C_DIS
LIN {X 0.043,Y -650.133,Z 867.423,A 0.000,B 0.000,C 90.000,E1 112.206} C_DIS
LIN {X 0.067,Y -645.868,Z 867.421,A 0.000,B 0.000,C 90.000,E1 111.844} C_DIS
LIN {X 0.241,Y -644.434,Z 867.421,A 0.000,B 0.000,C 90.000,E1 111.716} C_DIS
LIN {X -0.140,Y -642.738,Z 867.420,A 0.000,B 0.000,C 90.000,E1 111.642} C_DIS
LIN {X -0.001,Y -635.779,Z 867.418,A 0.000,B 0.000,C 90.000,E1 111.280} C_DIS
LIN {X 0.280,Y -624.282,Z 867.416,A 0.000,B 0.000,C 90.000,E1 110.791} C_DIS
LIN {X 0.206,Y -620.716,Z 867.415,A 0.000,B 0.000,C 90.000,E1 110.663} C_DIS
LIN {X -0.169,Y -607.291,Z 867.412,A 0.000,B 0.000,C 90.000,E1 110.120} C_DIS
LIN {X -0.087,Y -594.600,Z 867.408,A 0.000,B 0.000,C 90.000,E1 109.504} C_DIS
LIN {X -0.178,Y -588.018,Z 867.407,A 0.000,B 0.000,C 90.000,E1 109.214} C_DIS
LIN {X 0.202,Y -580.675,Z 867.405,A 0.000,B 0.000,C 90.000,E1 108.906} C_DIS
LIN {X -0.044,Y -566.311,Z 867.403,A 0.000,B 0.000,C 90.000,E1 108.489} C_DIS
LIN {X 0.127,Y -565.064,Z 867.402,A 0.000,B 0.000,C 90.000,E1 108.417} C_DIS
LIN {X 0.152,Y -562.083,Z 867.401,A 0.000,B 0.000,C 90.000,E1 108.236} C_DIS
LIN {X -0.016,Y -560.581,Z 867.400,A 0.000,B 0.000,C 90.000,E1 108.055} C_DIS
LIN {X -0.129,Y -560.028,Z 867.400,A 0.000,B 0.000,C 90.000,E1 107.928} C_DIS
LIN {X 0.002,Y -559.229,Z 867.398,A 0.000,B 0.000,C 90.000,E1 107.638} C_DIS
LIN {X -0.176,Y -558.740,Z 867.396,A 0.000,B 0.000,C 90.000,E1 107.221} C_DIS
LIN {X -0.089,Y -559.396,Z 867.377,A 0.000,B 0.000,C 90.000,E1 103.883} C_DIS
LIN {X -0.305,Y -560.228,Z 867.368,A 0.000,B 0.000,C 90.000,E1 102.243} C_DIS
LIN {X -0.196,Y -561.731,Z 867.356,A 0.000,B 0.000,C 90.000,E1 100.018} C_DIS
LIN {X 0.173,Y -562.329,Z 867.351,A 0.000,B 0.000,C 90.000,E1 99.151} C_DIS
LIN {X -0.170,Y -563.476,Z 867.342,A 0.000,B 0.000,C 90.000,E1 97.530} C_DIS
LIN {X -0.182,Y -564.140,Z 867.336,A 0.000,B 0.000,C 90.000,E1 96.429} C_DIS
LIN {X -0.009,Y -564.944,Z 867.326,A 0.000,B 0.000,C 90.000,E1 94.759} C_DIS
LIN {X 0.130,Y -565.559,Z 867.317,A 0.000,B 0.000,C 90.000,E1 93.094} C_DIS
LIN {X 0.253,Y -566.082,Z 867.308,A 0.000,B 0.000,C 90.000,E1 91.432} C_DIS
LIN {X 0.148,Y -566.358,Z 867.302,A 0.000,B 0.000,C 90.000,E1 90.344} C_DIS
LIN {X 0.166,Y -566.730,Z 867.294,A 0.000,B 0.000,C 90.000,E1 88.969} C_DIS
LIN {X -0.134,Y -567.048,Z 867.284,A 0.000,B 0.000,C 90.000,E1 87.078} C_DIS
LIN {X 0.052,Y -567.329,Z 867.275,A 0.000,B 0.000,C 90.000,E1 85.412} C_DIS
LIN {X 0.025,Y -567.532,Z 867.268,A 0.000,B 0.000,C 90.000,E1 84.318} C_DIS
LIN {X 0.172,Y -567.786,Z 867.261,A 0.000,B 0.000,C 90.000,E1 82.932} C_DIS
LIN {X 0.208,Y -568.422,Z 867.249,A 0.000,B 0.000,C 90.000,E1 80.735} C_DIS
LIN {X 0.072,Y -568.974,Z 867.240,A 0.000,B 0.000,C 90.000,E1 79.106} C_DIS
LIN {X 0.244,Y -569.824,Z 867.229,A 0.000,B 0.000,C 90.000,E1 77.173} C_DIS
LIN {X 0.055,Y -570.298,Z 867.221,A 0.000,B 0.000,C 90.000,E1 75.825} C_DIS
LIN {X -0.028,Y -570.963,Z 867.211,A 0.000,B 0.000,C 90.000,E1 73.921} C_DIS
LIN {X -0.277,Y -571.227,Z 867.202,A 0.000,B 0.000,C 90.000,E1 72.308} C_DIS
LIN {X -0.326,Y -571.340,Z 867.196,A 0.000,B 0.000,C 90.000,E1 71.221} C_DIS
LIN {X -0.205,Y -571.453,Z 867.186,A 0.000,B 0.000,C 90.000,E1 69.571} C_DIS
LIN {X -0.084,Y -571.446,Z 867.177,A 0.000,B 0.000,C 90.000,E1 67.922} C_DIS
LIN {X -0.055,Y -571.493,Z 867.168,A 0.000,B 0.000,C 90.000,E1 66.282} C_DIS
LIN {X -0.254,Y -571.332,Z 867.159,A 0.000,B 0.000,C 90.000,E1 64.665} C_DIS
LIN {X 0.190,Y -571.026,Z 867.152,A 0.000,B 0.000,C 90.000,E1 63.256} C_DIS
LIN {X 0.122,Y -570.681,Z 867.144,A 0.000,B 0.000,C 90.000,E1 61.897} C_DIS
LIN {X 0.041,Y -570.134,Z 867.136,A 0.000,B 0.000,C 90.000,E1 60.539} C_DIS
LIN {X -0.199,Y -569.799,Z 867.132,A 0.000,B 0.000,C 90.000,E1 59.744} C_DIS
LIN {X 0.086,Y -568.585,Z 867.123,A 0.000,B 0.000,C 90.000,E1 58.074} C_DIS
LIN {X 0.128,Y -567.906,Z 867.118,A 0.000,B 0.000,C 90.000,E1 57.248} C_DIS
LIN {X 0.052,Y -567.420,Z 867.115,A 0.000,B 0.000,C 90.000,E1 56.707} C_DIS
LIN {X 0.200,Y -566.147,Z 867.109,A 0.000,B 0.000,C 90.000,E1 55.595} C_DIS
LIN {X -0.130,Y -564.674,Z 867.103,A 0.000,B 0.000,C 90.000,E1 54.529} C_DIS
LIN {X -0.022,Y -563.053,Z 867.097,A 0.000,B 0.000,C 90.000,E1 53.417} C_DIS
LIN {X 0.291,Y -561.682,Z 867.092,A 0.000,B 0.000,C 90.000,E1 52.557} C_DIS
LIN {X 0.145,Y -560.141,Z 867.088,A 0.000,B 0.000,C 90.000,E1 51.743} C_DIS
LIN {X -0.013,Y -558.407,Z 867.083,A 0.000,B 0.000,C 90.000,E1 50.928} C_DIS
LIN {X 0.239,Y -556.364,Z 867.078,A 0.000,B 0.000,C 90.000,E1 50.070} C_DIS
LIN {X 0.035,Y -553.975,Z 867.074,A 0.000,B 0.000,C 90.000,E1 49.256} C_DIS
LIN {X 0.110,Y -552.288,Z 867.071,A 0.000,B 0.000,C 90.000,E1 48.690} C_DIS
LIN {X -0.139,Y -549.403,Z 867.066,A 0.000,B 0.000,C 90.000,E1 47.877} C_DIS
LIN {X -0.088,Y -547.301,Z 867.063,A 0.000,B 0.000,C 90.000,E1 47.310} C_DIS
LIN {X -0.025,Y -543.850,Z 867.058,A 0.000,B 0.000,C 90.000,E1 46.458} C_DIS
LIN {X 0.180,Y -540.691,Z 867.054,A 0.000,B 0.000,C 90.000,E1 45.729} C_DIS
LIN {X 0.170,Y -537.892,Z 867.051,A 0.000,B 0.000,C 90.000,E1 45.162} C_DIS
LIN {X 0.140,Y -534.859,Z 867.048,A 0.000,B 0.000,C 90.000,E1 44.595} C_DIS
LIN {X 0.258,Y -530.677,Z 867.044,A 0.000,B 0.000,C 90.000,E1 43.866} C_DIS
LIN {X 0.173,Y -527.060,Z 867.041,A 0.000,B 0.000,C 90.000,E1 43.299} C_DIS
LIN {X -0.095,Y -524.262,Z 867.038,A 0.000,B 0.000,C 90.000,E1 42.894} C_DIS
LIN {X 0.155,Y -520.204,Z 867.035,A 0.000,B 0.000,C 90.000,E1 42.285} C_DIS
LIN {X 0.031,Y -515.908,Z 867.032,A 0.000,B 0.000,C 90.000,E1 41.714} C_DIS
LIN {X -0.068,Y -511.397,Z 867.029,A 0.000,B 0.000,C 90.000,E1 41.148} C_DIS
LIN {X -0.014,Y -503.954,Z 867.024,A 0.000,B 0.000,C 90.000,E1 40.253} C_DIS
LIN {X 0.167,Y -498.621,Z 867.020,A 0.000,B 0.000,C 90.000,E1 39.644} C_DIS
LIN {X 0.007,Y -493.249,Z 867.017,A 0.000,B 0.000,C 90.000,E1 39.116} C_DIS
LIN {X 0.062,Y -487.932,Z 867.014,A 0.000,B 0.000,C 90.000,E1 38.588} C_DIS
LIN {X 0.011,Y -482.074,Z 867.011,A 0.000,B 0.000,C 90.000,E1 38.051} C_DIS
LIN {X 0.042,Y -477.565,Z 867.009,A 0.000,B 0.000,C 90.000,E1 37.649} C_DIS
LIN {X 0.143,Y -468.567,Z 867.005,A 0.000,B 0.000,C 90.000,E1 36.870} C_DIS
LIN {X 0.062,Y -456.101,Z 866.999,A 0.000,B 0.000,C 90.000,E1 35.884} C_DIS
LIN {X -0.195,Y -441.953,Z 866.993,A 0.000,B 0.000,C 90.000,E1 34.818} C_DIS
LIN {X 0.157,Y -418.891,Z 866.983,A 0.000,B 0.000,C 90.000,E1 32.880} C_DIS
LIN {X 0.166,Y -406.980,Z 866.977,A 0.000,B 0.000,C 90.000,E1 31.799} C_DIS
LIN {X -0.027,Y -401.309,Z 866.974,A 0.000,B 0.000,C 90.000,E1 31.258} C_DIS
LIN {X 0.140,Y -396.560,Z 866.971,A 0.000,B 0.000,C 90.000,E1 30.669} C_DIS
LIN {X -0.212,Y -393.787,Z 866.968,A 0.000,B 0.000,C 90.000,E1 30.335} C_DIS
LIN {X 0.094,Y -393.322,Z 866.968,A 0.000,B 0.000,C 90.000,E1 30.207} C_DIS
LIN {X 0.027,Y -391.992,Z 866.966,A 0.000,B 0.000,C 90.000,E1 29.873} C_DIS
LIN {X -0.077,Y -390.986,Z 866.965,A 0.000,B 0.000,C 90.000,E1 29.667} C_DIS
LIN {X -0.070,Y -389.826,Z 866.961,A 0.000,B 0.000,C 90.000,E1 28.999} C_DIS
LIN {X -0.002,Y -389.481,Z 866.958,A 0.000,B 0.000,C 90.000,E1 28.437} C_DIS
LIN {X 0.064,Y -389.907,Z 866.950,A 0.000,B 0.000,C 90.000,E1 27.001} C_DIS
LIN {X -0.076,Y -392.433,Z 866.930,A 0.000,B 0.000,C 90.000,E1 23.462} C_DIS
LIN {X 0.102,Y -395.466,Z 866.913,A 0.000,B 0.000,C 90.000,E1 20.248} C_DIS
LIN {X -0.027,Y -398.915,Z 866.895,A 0.000,B 0.000,C 90.000,E1 17.094} C_DIS
LIN {X -0.076,Y -401.987,Z 866.881,A 0.000,B 0.000,C 90.000,E1 14.647} C_DIS
LIN {X 0.149,Y -405.870,Z 866.866,A 0.000,B 0.000,C 90.000,E1 11.827} C_DIS
LIN {X -0.102,Y -409.074,Z 866.854,A 0.000,B 0.000,C 90.000,E1 9.782} C_DIS
LIN {X 0.048,Y -414.220,Z 866.837,A 0.000,B 0.000,C 90.000,E1 6.663} C_DIS
LIN {X -0.191,Y -417.956,Z 866.826,A 0.000,B 0.000,C 90.000,E1 4.645} C_DIS
LIN {X 0.086,Y -423.425,Z 866.811,A 0.000,B 0.000,C 90.000,E1 1.892} C_DIS
LIN {X -0.135,Y -429.792,Z 866.795,A 0.000,B 0.000,C 90.000,E1 359.141} C_DIS
LIN {X 0.110,Y -436.320,Z 866.780,A 0.000,B 0.000,C 90.000,E1 356.445} C_DIS
LIN {X -0.212,Y -440.636,Z 866.771,A 0.000,B 0.000,C 90.000,E1 354.837} C_DIS
LIN {X 0.040,Y -442.934,Z 866.768,A 0.000,B 0.000,C 90.000,E1 354.147} C_DIS
LIN {X 0.198,Y -444.242,Z 866.766,A 0.000,B 0.000,C 90.000,E1 353.799} C_DIS
LIN {X -0.129,Y -446.102,Z 866.764,A 0.000,B 0.000,C 90.000,E1 353.514} C_DIS
LIN {X -0.233,Y -450.062,Z 866.762,A 0.000,B 0.000,C 90.000,E1 353.109} C_DIS
LIN {X -0.137,Y -456.028,Z 866.759,A 0.000,B 0.000,C 90.000,E1 352.704} C_DIS
LIN {X 0.130,Y -470.153,Z 866.756,A 0.000,B 0.000,C 90.000,E1 352.008} C_DIS
LIN {X -0.263,Y -476.933,Z 866.754,A 0.000,B 0.000,C 90.000,E1 351.724} C_DIS
LIN {X 0.214,Y -486.676,Z 866.751,A 0.000,B 0.000,C 90.000,E1 351.141} C_DIS
LIN {X -0.252,Y -496.381,Z 866.748,A 0.000,B 0.000,C 90.000,E1 350.622} C_DIS
LIN {X -0.155,Y -508.932,Z 866.743,A 0.000,B 0.000,C 90.000,E1 349.803} C_DIS
LIN {X -0.124,Y -516.780,Z 866.740,A 0.000,B 0.000,C 90.000,E1 349.275} C_DIS
LIN {X -0.192,Y -525.961,Z 866.737,A 0.000,B 0.000,C 90.000,E1 348.634} C_DIS
LIN {X -0.004,Y -533.426,Z 866.734,A 0.000,B 0.000,C 90.000,E1 348.049} C_DIS
LIN {X -0.116,Y -542.081,Z 866.730,A 0.000,B 0.000,C 90.000,E1 347.353} C_DIS
LIN {X 0.139,Y -550.381,Z 866.726,A 0.000,B 0.000,C 90.000,E1 346.589} C_DIS
LIN {X 0.033,Y -558.264,Z 866.721,A 0.000,B 0.000,C 90.000,E1 345.825} C_DIS
LIN {X -0.102,Y -564.583,Z 866.718,A 0.000,B 0.000,C 90.000,E1 345.172} C_DIS
LIN {X 0.101,Y -571.782,Z 866.713,A 0.000,B 0.000,C 90.000,E1 344.338} C_DIS
LIN {X -0.281,Y -578.381,Z 866.709,A 0.000,B 0.000,C 90.000,E1 343.559} C_DIS
LIN {X -0.040,Y -584.520,Z 866.704,A 0.000,B 0.000,C 90.000,E1 342.725} C_DIS
LIN {X -0.297,Y -590.055,Z 866.700,A 0.000,B 0.000,C 90.000,E1 341.945} C_DIS
LIN {X 0.251,Y -595.288,Z 866.695,A 0.000,B 0.000,C 90.000,E1 341.094} C_DIS
LIN {X 0.003,Y -601.548,Z 866.689,A 0.000,B 0.000,C 90.000,E1 340.061} C_DIS
LIN {X -0.167,Y -607.438,Z 866.683,A 0.000,B 0.000,C 90.000,E1 339.028} C_DIS
LIN {X -0.097,Y -615.133,Z 866.676,A 0.000,B 0.000,C 90.000,E1 337.592} C_DIS
LIN {X 0.167,Y -618.426,Z 866.672,A 0.000,B 0.000,C 90.000,E1 336.922} C_DIS
LIN {X -0.120,Y -622.268,Z 866.668,A 0.000,B 0.000,C 90.000,E1 336.177} C_DIS
LIN {X -0.114,Y -626.362,Z 866.663,A 0.000,B 0.000,C 90.000,E1 335.281} C_DIS
LIN {X -0.337,Y -629.779,Z 866.658,A 0.000,B 0.000,C 90.000,E1 334.537} C_DIS
LIN {X -0.224,Y -633.959,Z 866.653,A 0.000,B 0.000,C 90.000,E1 333.512} C_DIS
LIN {X -0.052,Y -637.912,Z 866.647,A 0.000,B 0.000,C 90.000,E1 332.487} C_DIS
LIN {X 0.109,Y -640.650,Z 866.643,A 0.000,B 0.000,C 90.000,E1 331.719} C_DIS
LIN {X 0.180,Y -644.930,Z 866.636,A 0.000,B 0.000,C 90.000,E1 330.461} C_DIS
LIN {X 0.330,Y -649.049,Z 866.629,A 0.000,B 0.000,C 90.000,E1 329.203} C_DIS
LIN {X -0.015,Y -652.749,Z 866.622,A 0.000,B 0.000,C 90.000,E1 327.995} C_DIS
LIN {X 0.056,Y -654.795,Z 866.618,A 0.000,B 0.000,C 90.000,E1 327.248} C_DIS
LIN {X -0.306,Y -657.381,Z 866.613,A 0.000,B 0.000,C 90.000,E1 326.294} C_DIS
LIN {X -0.267,Y -659.701,Z 866.607,A 0.000,B 0.000,C 90.000,E1 325.308} C_DIS
LIN {X -0.096,Y -662.164,Z 866.600,A 0.000,B 0.000,C 90.000,E1 324.069} C_DIS
LIN {X 0.001,Y -663.917,Z 866.595,A 0.000,B 0.000,C 90.000,E1 323.084} C_DIS
LIN {X 0.084,Y -665.788,Z 866.588,A 0.000,B 0.000,C 90.000,E1 321.859} C_DIS
LIN {X -0.338,Y -667.774,Z 866.580,A 0.000,B 0.000,C 90.000,E1 320.436} C_DIS
LIN {X -0.281,Y -669.173,Z 866.573,A 0.000,B 0.000,C 90.000,E1 319.218} C_DIS
LIN {X -0.203,Y -670.239,Z 866.568,A 0.000,B 0.000,C 90.000,E1 318.243} C_DIS
LIN {X -0.065,Y -672.370,Z 866.557,A 0.000,B 0.000,C 90.000,E1 316.296} C_DIS
LIN {X 0.014,Y -673.640,Z 866.552,A 0.000,B 0.000,C 90.000,E1 315.324} C_DIS
LIN {X 0.086,Y -674.388,Z 866.548,A 0.000,B 0.000,C 90.000,E1 314.595} C_DIS
LIN {X -0.132,Y -676.423,Z 866.536,A 0.000,B 0.000,C 90.000,E1 312.447} C_DIS
LIN {X 0.068,Y -677.598,Z 866.529,A 0.000,B 0.000,C 90.000,E1 311.229} C_DIS
LIN {X 0.287,Y -678.659,Z 866.522,A 0.000,B 0.000,C 90.000,E1 310.011} C_DIS
LIN {X 0.110,Y -679.889,Z 866.514,A 0.000,B 0.000,C 90.000,E1 308.588} C_DIS
LIN {X -0.326,Y -681.253,Z 866.505,A 0.000,B 0.000,C 90.000,E1 306.950} C_DIS
LIN {X -0.338,Y -682.338,Z 866.497,A 0.000,B 0.000,C 90.000,E1 305.518} C_DIS
LIN {X -0.169,Y -683.264,Z 866.489,A 0.000,B 0.000,C 90.000,E1 304.072} C_DIS
LIN {X -0.166,Y -684.763,Z 866.477,A 0.000,B 0.000,C 90.000,E1 301.926} C_DIS
LIN {X -0.113,Y -686.046,Z 866.468,A 0.000,B 0.000,C 90.000,E1 300.256} C_DIS
LIN {X 0.303,Y -688.190,Z 866.455,A 0.000,B 0.000,C 90.000,E1 297.847} C_DIS
LIN {X 0.154,Y -689.641,Z 866.447,A 0.000,B 0.000,C 90.000,E1 296.437} C_DIS
LIN {X 0.031,Y -691.123,Z 866.439,A 0.000,B 0.000,C 90.000,E1 295.027} C_DIS
LIN {X 0.068,Y -691.905,Z 866.434,A 0.000,B 0.000,C 90.000,E1 294.079} C_DIS
LIN {X -0.128,Y -692.087,Z 866.430,A 0.000,B 0.000,C 90.000,E1 293.387} C_DIS
LIN {X 0.076,Y -691.471,Z 866.427,A 0.000,B 0.000,C 90.000,E1 292.898} C_DIS
LIN {X 0.311,Y -691.031,Z 866.426,A 0.000,B 0.000,C 90.000,E1 292.642} C_DIS
LIN {X -0.358,Y -689.961,Z 866.425,A 0.000,B 0.000,C 90.000,E1 292.461} C_DIS
LIN {X -0.015,Y -687.865,Z 866.423,A 0.000,B 0.000,C 90.000,E1 292.078} C_DIS
LIN {X -0.161,Y -687.073,Z 866.422,A 0.000,B 0.000,C 90.000,E1 291.972} C_DIS
LIN {X -0.052,Y -685.996,Z 866.421,A 0.000,B 0.000,C 90.000,E1 291.844} C_DIS
LIN {X 0.056,Y -684.361,Z 866.421,A 0.000,B 0.000,C 90.000,E1 291.716} C_DIS
LIN {X 0.353,Y -678.841,Z 866.419,A 0.000,B 0.000,C 90.000,E1 291.408} C_DIS
LIN {X 0.020,Y -677.070,Z 866.419,A 0.000,B 0.000,C 90.000,E1 291.354} C_DIS
LIN {X 0.115,Y -675.322,Z 866.418,A 0.000,B 0.000,C 90.000,E1 291.280} C_DIS
LIN {X 0.317,Y -669.931,Z 866.417,A 0.000,B 0.000,C 90.000,E1 291.099} C_DIS
LIN {X -0.094,Y -659.040,Z 866.416,A 0.000,B 0.000,C 90.000,E1 290.865} C_DIS
LIN {X -0.309,Y -655.814,Z 866.415,A 0.000,B 0.000,C 90.000,E1 290.791} C_DIS
LIN {X 0.218,Y -651.156,Z 866.414,A 0.000,B 0.000,C 90.000,E1 290.556} C_DIS
LIN {X 0.054,Y -648.335,Z 866.413,A 0.000,B 0.000,C 90.000,E1 290.375} C_DIS
LIN {X 0.016,Y -648.311,Z 866.413,A 0.000,B 0.000,C 90.000,E1 290.375} C_DIS
LIN {X 0.116,Y -647.556,Z 866.412,A 0.000,B 0.000,C 90.000,E1 290.194} C_DIS
LIN {X 0.071,Y -647.555,Z 866.412,A 0.000,B 0.000,C 90.000,E1 290.194} C_DIS
LIN {X 0.231,Y -648.072,Z 866.411,A 0.000,B 0.000,C 90.000,E1 289.939} C_DIS
LIN {X -0.294,Y -650.276,Z 866.408,A 0.000,B 0.000,C 90.000,E1 289.450} C_DIS
LIN {X 0.121,Y -657.547,Z 866.400,A 0.000,B 0.000,C 90.000,E1 288.055} C_DIS
LIN {X -0.061,Y -660.517,Z 866.397,A 0.000,B 0.000,C 90.000,E1 287.457} C_DIS
LIN {X -0.173,Y -663.704,Z 866.393,A 0.000,B 0.000,C 90.000,E1 286.732} C_DIS
LIN {X 0.194,Y -666.336,Z 866.389,A 0.000,B 0.000,C 90.000,E1 285.969} C_DIS
LIN {X 0.211,Y -667.869,Z 866.386,A 0.000,B 0.000,C 90.000,E1 285.481} C_DIS
LIN {X -0.017,Y -669.745,Z 866.382,A 0.000,B 0.000,C 90.000,E1 284.773} C_DIS
LIN {X -0.225,Y -671.114,Z 866.378,A 0.000,B 0.000,C 90.000,E1 284.064} C_DIS
LIN {X 0.297,Y -671.875,Z 866.375,A 0.000,B 0.000,C 90.000,E1 283.536} C_DIS
LIN {X 0.110,Y -672.652,Z 866.371,A 0.000,B 0.000,C 90.000,E1 282.827} C_DIS
LIN {X -0.073,Y -673.192,Z 866.367,A 0.000,B 0.000,C 90.000,E1 282.119} C_DIS
LIN {X 0.269,Y -673.325,Z 866.363,A 0.000,B 0.000,C 90.000,E1 281.366} C_DIS
LIN {X 0.147,Y -673.157,Z 866.361,A 0.000,B 0.000,C 90.000,E1 280.894} C_DIS
LIN {X -0.103,Y -672.735,Z 866.358,A 0.000,B 0.000,C 90.000,E1 280.433} C_DIS
LIN {X -0.232,Y -672.061,Z 866.355,A 0.000,B 0.000,C 90.000,E1 279.962} C_DIS
LIN {X 0.180,Y -671.125,Z 866.353,A 0.000,B 0.000,C 90.000,E1 279.443} C_DIS
LIN {X 0.108,Y -670.605,Z 866.351,A 0.000,B 0.000,C 90.000,E1 279.208} C_DIS
LIN {X -0.147,Y -669.172,Z 866.349,A 0.000,B 0.000,C 90.000,E1 278.746} C_DIS
LIN {X 0.349,Y -667.450,Z 866.346,A 0.000,B 0.000,C 90.000,E1 278.219} C_DIS
LIN {X 0.075,Y -665.433,Z 866.343,A 0.000,B 0.000,C 90.000,E1 277.757} C_DIS
LIN {X -0.209,Y -663.095,Z 866.340,A 0.000,B 0.000,C 90.000,E1 277.296} C_DIS
LIN {X 0.246,Y -661.189,Z 866.338,A 0.000,B 0.000,C 90.000,E1 276.891} C_DIS
LIN {X -0.067,Y -658.289,Z 866.336,A 0.000,B 0.000,C 90.000,E1 276.429} C_DIS
LIN {X 0.252,Y -654.995,Z 866.333,A 0.000,B 0.000,C 90.000,E1 275.910} C_DIS
LIN {X -0.163,Y -651.138,Z 866.330,A 0.000,B 0.000,C 90.000,E1 275.454} C_DIS
LIN {X -0.001,Y -645.477,Z 866.327,A 0.000,B 0.000,C 90.000,E1 274.821} C_DIS
LIN {X -0.068,Y -639.430,Z 866.324,A 0.000,B 0.000,C 90.000,E1 274.245} C_DIS
LIN {X -0.098,Y -633.968,Z 866.321,A 0.000,B 0.000,C 90.000,E1 273.784} C_DIS
LIN {X 0.253,Y -630.006,Z 866.319,A 0.000,B 0.000,C 90.000,E1 273.440} C_DIS
LIN {X 0.078,Y -624.194,Z 866.317,A 0.000,B 0.000,C 90.000,E1 273.037} C_DIS
LIN {X 0.078,Y -617.918,Z 866.315,A 0.000,B 0.000,C 90.000,E1 272.636} C_DIS
LIN {X -0.220,Y -611.310,Z 866.313,A 0.000,B 0.000,C 90.000,E1 272.293} C_DIS
LIN {X -0.132,Y -604.592,Z 866.311,A 0.000,B 0.000,C 90.000,E1 271.949} C_DIS
LIN {X -0.283,Y -597.435,Z 866.309,A 0.000,B 0.000,C 90.000,E1 271.661} C_DIS
LIN {X -0.035,Y -590.052,Z 866.308,A 0.000,B 0.000,C 90.000,E1 271.375} C_DIS
LIN {X -0.048,Y -584.132,Z 866.307,A 0.000,B 0.000,C 90.000,E1 271.203} C_DIS
LIN {X -0.024,Y -576.367,Z 866.306,A 0.000,B 0.000,C 90.000,E1 271.031} C_DIS
LIN {X 0.189,Y -570.943,Z 866.305,A 0.000,B 0.000,C 90.000,E1 270.917} C_DIS
LIN {X 0.016,Y -563.616,Z 866.305,A 0.000,B 0.000,C 90.000,E1 270.859} C_DIS
LIN {X 0.131,Y -553.985,Z 866.305,A 0.000,B 0.000,C 90.000,E1 270.802} C_DIS
LIN {X -0.007,Y -552.372,Z 866.305,A 0.000,B 0.000,C 90.000,E1 270.802} C_DIS
LIN {X -0.207,Y -549.663,Z 866.304,A 0.000,B 0.000,C 90.000,E1 270.745} C_DIS
LIN {X -0.241,Y -549.565,Z 866.304,A 0.000,B 0.000,C 90.000,E1 270.745} C_DIS
LIN {X -0.138,Y -547.670,Z 866.303,A 0.000,B 0.000,C 90.000,E1 270.516} C_DIS
LIN {X 0.014,Y -546.693,Z 866.301,A 0.000,B 0.000,C 90.000,E1 270.115} C_DIS
LIN {X 0.104,Y -545.734,Z 866.298,A 0.000,B 0.000,C 90.000,E1 269.542} C_DIS
LIN {X -0.043,Y -543.197,Z 866.282,A 0.000,B 0.000,C 90.000,E1 266.731} C_DIS
LIN {X 0.115,Y -542.294,Z 866.274,A 0.000,B 0.000,C 90.000,E1 265.298} C_DIS
LIN {X -0.195,Y -541.323,Z 866.266,A 0.000,B 0.000,C 90.000,E1 263.913} C_DIS
LIN {X 0.024,Y -540.178,Z 866.258,A 0.000,B 0.000,C 90.000,E1 262.470} C_DIS
LIN {X 0.214,Y -538.877,Z 866.250,A 0.000,B 0.000,C 90.000,E1 261.027} C_DIS
LIN {X -0.013,Y -537.240,Z 866.241,A 0.000,B 0.000,C 90.000,E1 259.342} C_DIS
LIN {X -0.234,Y -535.708,Z 866.233,A 0.000,B 0.000,C 90.000,E1 257.937} C_DIS
LIN {X 0.108,Y -534.367,Z 866.227,A 0.000,B 0.000,C 90.000,E1 256.756} C_DIS
LIN {X -0.037,Y -532.626,Z 866.219,A 0.000,B 0.000,C 90.000,E1 255.338} C_DIS
LIN {X 0.260,Y -531.245,Z 866.212,A 0.000,B 0.000,C 90.000,E1 254.157} C_DIS
LIN {X -0.136,Y -529.194,Z 866.203,A 0.000,B 0.000,C 90.000,E1 252.472} C_DIS
LIN {X 0.249,Y -527.816,Z 866.196,A 0.000,B 0.000,C 90.000,E1 251.275} C_DIS
LIN {X -0.222,Y -525.900,Z 866.188,A 0.000,B 0.000,C 90.000,E1 249.880} C_DIS
LIN {X -0.055,Y -523.918,Z 866.180,A 0.000,B 0.000,C 90.000,E1 248.411} C_DIS
LIN {X -0.058,Y -521.336,Z 866.170,A 0.000,B 0.000,C 90.000,E1 246.666} C_DIS
LIN {X 0.067,Y -519.536,Z 866.164,A 0.000,B 0.000,C 90.000,E1 245.485} C_DIS
LIN {X 0.173,Y -516.827,Z 866.154,A 0.000,B 0.000,C 90.000,E1 243.717} C_DIS
LIN {X -0.018,Y -513.812,Z 866.144,A 0.000,B 0.000,C 90.000,E1 241.975} C_DIS
LIN {X -0.031,Y -510.730,Z 866.135,A 0.000,B 0.000,C 90.000,E1 240.205} C_DIS
LIN {X 0.179,Y -508.546,Z 866.128,A 0.000,B 0.000,C 90.000,E1 238.997} C_DIS
LIN {X -0.019,Y -505.716,Z 866.120,A 0.000,B 0.000,C 90.000,E1 237.533} C_DIS
LIN {X 0.273,Y -502.793,Z 866.111,A 0.000,B 0.000,C 90.000,E1 236.008} C_DIS
LIN {X 0.054,Y -500.902,Z 866.106,A 0.000,B 0.000,C 90.000,E1 235.135} C_DIS
LIN {X 0.261,Y -498.105,Z 866.100,A 0.000,B 0.000,C 90.000,E1 233.909} C_DIS
LIN {X 0.157,Y -493.716,Z 866.090,A 0.000,B 0.000,C 90.000,E1 232.110} C_DIS
LIN {X 0.106,Y -490.121,Z 866.081,A 0.000,B 0.000,C 90.000,E1 230.598} C_DIS
LIN {X -0.085,Y -486.661,Z 866.073,A 0.000,B 0.000,C 90.000,E1 229.094} C_DIS
LIN {X 0.054,Y -481.221,Z 866.059,A 0.000,B 0.000,C 90.000,E1 226.620} C_DIS
LIN {X 0.118,Y -477.188,Z 866.049,A 0.000,B 0.000,C 90.000,E1 224.757} C_DIS
LIN {X -0.220,Y -475.143,Z 866.044,A 0.000,B 0.000,C 90.000,E1 223.866} C_DIS
LIN {X 0.041,Y -471.097,Z 866.033,A 0.000,B 0.000,C 90.000,E1 221.962} C_DIS
LIN {X -0.071,Y -467.024,Z 866.023,A 0.000,B 0.000,C 90.000,E1 220.092} C_DIS
LIN {X -0.156,Y -462.310,Z 866.010,A 0.000,B 0.000,C 90.000,E1 217.890} C_DIS
LIN {X -0.015,Y -458.311,Z 866.000,A 0.000,B 0.000,C 90.000,E1 215.964} C_DIS
LIN {X 0.039,Y -454.903,Z 865.991,A 0.000,B 0.000,C 90.000,E1 214.358} C_DIS
LIN {X -0.097,Y -449.387,Z 865.977,A 0.000,B 0.000,C 90.000,E1 211.799} C_DIS
LIN {X 0.286,Y -445.925,Z 865.968,A 0.000,B 0.000,C 90.000,E1 210.129} C_DIS
LIN {X -0.173,Y -441.825,Z 865.957,A 0.000,B 0.000,C 90.000,E1 208.231} C_DIS
LIN {X -0.112,Y -436.980,Z 865.944,A 0.000,B 0.000,C 90.000,E1 205.924} C_DIS
LIN {X -0.194,Y -432.770,Z 865.933,A 0.000,B 0.000,C 90.000,E1 203.951} C_DIS
LIN {X -0.142,Y -429.405,Z 865.924,A 0.000,B 0.000,C 90.000,E1 202.280} C_DIS
LIN {X 0.045,Y -426.681,Z 865.916,A 0.000,B 0.000,C 90.000,E1 200.918} C_DIS
LIN {X 0.011,Y -422.699,Z 865.905,A 0.000,B 0.000,C 90.000,E1 198.906} C_DIS
LIN {X -0.026,Y -419.442,Z 865.896,A 0.000,B 0.000,C 90.000,E1 197.221} C_DIS
LIN {X 0.111,Y -416.708,Z 865.888,A 0.000,B 0.000,C 90.000,E1 195.843} C_DIS
LIN {X 0.232,Y -413.247,Z 865.879,A 0.000,B 0.000,C 90.000,E1 194.120} C_DIS
LIN {X -0.154,Y -407.820,Z 865.863,A 0.000,B 0.000,C 90.000,E1 191.422} C_DIS
LIN {X -0.013,Y -405.075,Z 865.856,A 0.000,B 0.000,C 90.000,E1 190.018} C_DIS
LIN {X 0.009,Y -402.355,Z 865.848,A 0.000,B 0.000,C 90.000,E1 188.624} C_DIS
LIN {X 0.100,Y -395.661,Z 865.828,A 0.000,B 0.000,C 90.000,E1 185.106} C_DIS
LIN {X 0.047,Y -388.973,Z 865.805,A 0.000,B 0.000,C 90.000,E1 180.859} C_DIS
LIN {X -0.022,Y -386.500,Z 865.795,A 0.000,B 0.000,C 90.000,E1 179.083} C_DIS
LIN {X -0.134,Y -383.956,Z 865.785,A 0.000,B 0.000,C 90.000,E1 177.306} C_DIS
LIN {X 0.102,Y -381.374,Z 865.775,A 0.000,B 0.000,C 90.000,E1 175.469} C_DIS
LIN {X -0.135,Y -376.986,Z 865.757,A 0.000,B 0.000,C 90.000,E1 172.243} C_DIS
LIN {X 0.079,Y -375.030,Z 865.747,A 0.000,B 0.000,C 90.000,E1 170.387} C_DIS
LIN {X 0.067,Y -373.684,Z 865.739,A 0.000,B 0.000,C 90.000,E1 168.926} C_DIS
LIN {X 0.114,Y -372.844,Z 865.724,A 0.000,B 0.000,C 90.000,E1 166.353} C_DIS
LIN {X -0.050,Y -372.945,Z 865.720,A 0.000,B 0.000,C 90.000,E1 165.644} C_DIS
LIN {X -0.085,Y -373.189,Z 865.718,A 0.000,B 0.000,C 90.000,E1 165.283} C_DIS
LIN {X 0.128,Y -373.393,Z 865.715,A 0.000,B 0.000,C 90.000,E1 164.700} C_DIS
LIN {X 0.082,Y -374.071,Z 865.712,A 0.000,B 0.000,C 90.000,E1 164.157} C_DIS
LIN {X 0.068,Y -374.244,Z 865.711,A 0.000,B 0.000,C 90.000,E1 163.976} C_DIS
LIN {X -0.055,Y -375.105,Z 865.709,A 0.000,B 0.000,C 90.000,E1 163.559} C_DIS
LIN {X -0.079,Y -375.658,Z 865.707,A 0.000,B 0.000,C 90.000,E1 163.196} C_DIS
LIN {X 0.004,Y -377.783,Z 865.702,A 0.000,B 0.000,C 90.000,E1 162.362} C_DIS
LIN {X 0.111,Y -380.089,Z 865.700,A 0.000,B 0.000,C 90.000,E1 161.891} C_DIS
LIN {X -0.066,Y -383.005,Z 865.697,A 0.000,B 0.000,C 90.000,E1 161.456} C_DIS
LIN {X -0.064,Y -384.384,Z 865.696,A 0.000,B 0.000,C 90.000,E1 161.275} C_DIS
LIN {X 0.049,Y -390.839,Z 865.693,A 0.000,B 0.000,C 90.000,E1 160.678} C_DIS
LIN {X -0.115,Y -396.871,Z 865.691,A 0.000,B 0.000,C 90.000,E1 160.369} C_DIS
LIN {X -0.044,Y -406.189,Z 865.689,A 0.000,B 0.000,C 90.000,E1 159.934} C_DIS
LIN {X 0.038,Y -411.300,Z 865.687,A 0.000,B 0.000,C 90.000,E1 159.699} C_DIS
LIN {X -0.072,Y -418.118,Z 865.685,A 0.000,B 0.000,C 90.000,E1 159.390} C_DIS
LIN {X 0.064,Y -427.944,Z 865.683,A 0.000,B 0.000,C 90.000,E1 158.847} C_DIS
LIN {X -0.141,Y -434.242,Z 865.680,A 0.000,B 0.000,C 90.000,E1 158.465} C_DIS
LIN {X 0.008,Y -443.430,Z 865.677,A 0.000,B 0.000,C 90.000,E1 157.794} C_DIS
LIN {X 0.054,Y -454.374,Z 865.672,A 0.000,B 0.000,C 90.000,E1 156.922} C_DIS
LIN {X -0.080,Y -461.439,Z 865.668,A 0.000,B 0.000,C 90.000,E1 156.282} C_DIS
LIN {X 0.100,Y -471.352,Z 865.663,A 0.000,B 0.000,C 90.000,E1 155.281} C_DIS
LIN {X 0.002,Y -476.851,Z 865.660,A 0.000,B 0.000,C 90.000,E1 154.717} C_DIS
LIN {X -0.017,Y -484.645,Z 865.655,A 0.000,B 0.000,C 90.000,E1 153.819} C_DIS
LIN {X 0.090,Y -490.830,Z 865.650,A 0.000,B 0.000,C 90.000,E1 153.050} C_DIS
LIN {X 0.269,Y -496.557,Z 865.646,A 0.000,B 0.000,C 90.000,E1 152.281} C_DIS
LIN {X -0.225,Y -500.092,Z 865.644,A 0.000,B 0.000,C 90.000,E1 151.897} C_DIS
LIN {X 0.051,Y -508.903,Z 865.637,A 0.000,B 0.000,C 90.000,E1 150.667} C_DIS
LIN {X 0.197,Y -512.080,Z 865.635,A 0.000,B 0.000,C 90.000,E1 150.205} C_DIS
LIN {X -0.248,Y -516.101,Z 865.631,A 0.000,B 0.000,C 90.000,E1 149.665} C_DIS
LIN {X -0.050,Y -519.254,Z 865.629,A 0.000,B 0.000,C 90.000,E1 149.203} C_DIS
LIN {X 0.130,Y -529.331,Z 865.620,A 0.000,B 0.000,C 90.000,E1 147.582} C_DIS
LIN {X 0.222,Y -534.357,Z 865.615,A 0.000,B 0.000,C 90.000,E1 146.707} C_DIS
LIN {X 0.073,Y -540.014,Z 865.610,A 0.000,B 0.000,C 90.000,E1 145.722} C_DIS
LIN {X -0.030,Y -543.784,Z 865.606,A 0.000,B 0.000,C 90.000,E1 145.022} C_DIS
LIN {X -0.193,Y -549.735,Z 865.599,A 0.000,B 0.000,C 90.000,E1 143.909} C_DIS
LIN {X 0.206,Y -558.575,Z 865.590,A 0.000,B 0.000,C 90.000,E1 142.190} C_DIS
LIN {X -0.058,Y -561.496,Z 865.587,A 0.000,B 0.000,C 90.000,E1 141.662} C_DIS
LIN {X -0.092,Y -569.478,Z 865.579,A 0.000,B 0.000,C 90.000,E1 140.150} C_DIS
LIN {X -0.031,Y -572.977,Z 865.575,A 0.000,B 0.000,C 90.000,E1 139.461} C_DIS
LIN {X 0.038,Y -578.232,Z 865.569,A 0.000,B 0.000,C 90.000,E1 138.366} C_DIS
LIN {X 0.015,Y -588.722,Z 865.557,A 0.000,B 0.000,C 90.000,E1 136.215} C_DIS
LIN {X 0.120,Y -592.610,Z 865.552,A 0.000,B 0.000,C 90.000,E1 135.405} C_DIS
LIN {X 0.358,Y -598.252,Z 865.546,A 0.000,B 0.000,C 90.000,E1 134.190} C_DIS
LIN {X -0.057,Y -603.167,Z 865.540,A 0.000,B 0.000,C 90.000,E1 133.176} C_DIS
LIN {X 0.061,Y -610.169,Z 865.531,A 0.000,B 0.000,C 90.000,E1 131.595} C_DIS
LIN {X 0.251,Y -614.577,Z 865.525,A 0.000,B 0.000,C 90.000,E1 130.539} C_DIS
LIN {X -0.059,Y -619.709,Z 865.518,A 0.000,B 0.000,C 90.000,E1 129.277} C_DIS
LIN {X -0.132,Y -623.683,Z 865.513,A 0.000,B 0.000,C 90.000,E1 128.257} C_DIS
LIN {X -0.124,Y -631.132,Z 865.501,A 0.000,B 0.000,C 90.000,E1 126.217} C_DIS
LIN {X -0.282,Y -632.971,Z 865.498,A 0.000,B 0.000,C 90.000,E1 125.724} C_DIS
LIN {X -0.039,Y -636.291,Z 865.493,A 0.000,B 0.000,C 90.000,E1 124.692} C_DIS
LIN {X -0.275,Y -639.349,Z 865.487,A 0.000,B 0.000,C 90.000,E1 123.706} C_DIS
LIN {X 0.055,Y -642.128,Z 865.482,A 0.000,B 0.000,C 90.000,E1 122.673} C_DIS
LIN {X -0.382,Y -643.373,Z 865.479,A 0.000,B 0.000,C 90.000,E1 122.212} C_DIS
LIN {X 0.139,Y -646.629,Z 865.471,A 0.000,B 0.000,C 90.000,E1 120.669} C_DIS
LIN {X 0.142,Y -647.985,Z 865.466,A 0.000,B 0.000,C 90.000,E1 119.922} C_DIS
LIN {X -0.370,Y -650.774,Z 865.457,A 0.000,B 0.000,C 90.000,E1 118.231} C_DIS
LIN {X 0.029,Y -652.211,Z 865.451,A 0.000,B 0.000,C 90.000,E1 117.206} C_DIS
LIN {X -0.239,Y -653.228,Z 865.447,A 0.000,B 0.000,C 90.000,E1 116.488} C_DIS
LIN {X 0.191,Y -654.156,Z 865.442,A 0.000,B 0.000,C 90.000,E1 115.463} C_DIS
LIN {X -0.241,Y -654.760,Z 865.436,A 0.000,B 0.000,C 90.000,E1 114.515} C_DIS
LIN {X -0.132,Y -654.896,Z 865.435,A 0.000,B 0.000,C 90.000,E1 114.259} C_DIS
LIN {X -0.178,Y -654.595,Z 865.432,A 0.000,B 0.000,C 90.000,E1 113.770} C_DIS
LIN {X -0.069,Y -654.353,Z 865.431,A 0.000,B 0.000,C 90.000,E1 113.515} C_DIS
LIN {X -0.112,Y -652.733,Z 865.428,A 0.000,B 0.000,C 90.000,E1 113.025} C_DIS
LIN {X -0.009,Y -651.511,Z 865.427,A 0.000,B 0.000,C 90.000,E1 112.770} C_DIS
LIN {X 0.134,Y -649.005,Z 865.424,A 0.000,B 0.000,C 90.000,E1 112.386} C_DIS
LIN {X -0.067,Y -648.030,Z 865.424,A 0.000,B 0.000,C 90.000,E1 112.280} C_DIS
LIN {X 0.121,Y -642.446,Z 865.421,A 0.000,B 0.000,C 90.000,E1 111.791} C_DIS
LIN {X -0.130,Y -638.321,Z 865.420,A 0.000,B 0.000,C 90.000,E1 111.589} C_DIS
LIN {X 0.214,Y -633.090,Z 865.418,A 0.000,B 0.000,C 90.000,E1 111.280} C_DIS
LIN {X 0.346,Y -628.883,Z 865.417,A 0.000,B 0.000,C 90.000,E1 111.099} C_DIS
LIN {X 0.259,Y -626.201,Z 865.417,A 0.000,B 0.000,C 90.000,E1 110.972} C_DIS
LIN {X 0.020,Y -623.361,Z 865.416,A 0.000,B 0.000,C 90.000,E1 110.865} C_DIS
LIN {X -0.224,Y -619.512,Z 865.415,A 0.000,B 0.000,C 90.000,E1 110.737} C_DIS
LIN {X -0.219,Y -613.955,Z 865.414,A 0.000,B 0.000,C 90.000,E1 110.482} C_DIS
LIN {X -0.130,Y -607.248,Z 865.412,A 0.000,B 0.000,C 90.000,E1 110.174} C_DIS
LIN {X -0.277,Y -594.668,Z 865.409,A 0.000,B 0.000,C 90.000,E1 109.577} C_DIS
LIN {X -0.234,Y -587.831,Z 865.407,A 0.000,B 0.000,C 90.000,E1 109.268} C_DIS
LIN {X 0.116,Y -580.409,Z 865.405,A 0.000,B 0.000,C 90.000,E1 108.960} C_DIS
LIN {X -0.089,Y -566.161,Z 865.403,A 0.000,B 0.000,C 90.000,E1 108.544} C_DIS
LIN {X -0.210,Y -562.124,Z 865.402,A 0.000,B 0.000,C 90.000,E1 108.308} C_DIS
LIN {X 0.279,Y -560.712,Z 865.401,A 0.000,B 0.000,C 90.000,E1 108.055} C_DIS
LIN {X 0.103,Y -559.534,Z 865.398,A 0.000,B 0.000,C 90.000,E1 107.692} C_DIS
LIN {X 0.322,Y -558.947,Z 865.395,A 0.000,B 0.000,C 90.000,E1 107.094} C_DIS
LIN {X -0.038,Y -559.128,Z 865.384,A 0.000,B 0.000,C 90.000,E1 105.190} C_DIS
LIN {X 0.037,Y -560.311,Z 865.369,A 0.000,B 0.000,C 90.000,E1 102.411} C_DIS
LIN {X 0.037,Y -561.767,Z 865.357,A 0.000,B 0.000,C 90.000,E1 100.197} C_DIS
LIN {X 0.011,Y -562.564,Z 865.351,A 0.000,B 0.000,C 90.000,E1 99.095} C_DIS
LIN {X 0.152,Y -563.528,Z 865.343,A 0.000,B 0.000,C 90.000,E1 97.701} C_DIS
LIN {X 0.228,Y -564.360,Z 865.335,A 0.000,B 0.000,C 90.000,E1 96.315} C_DIS
LIN {X -0.052,Y -565.275,Z 865.325,A 0.000,B 0.000,C 90.000,E1 94.416} C_DIS
LIN {X 0.100,Y -565.865,Z 865.315,A 0.000,B 0.000,C 90.000,E1 92.751} C_DIS
LIN {X 0.234,Y -566.358,Z 865.306,A 0.000,B 0.000,C 90.000,E1 91.088} C_DIS
LIN {X 0.017,Y -566.566,Z 865.302,A 0.000,B 0.000,C 90.000,E1 90.286} C_DIS
LIN {X 0.037,Y -566.914,Z 865.294,A 0.000,B 0.000,C 90.000,E1 88.912} C_DIS
LIN {X -0.258,Y -567.237,Z 865.283,A 0.000,B 0.000,C 90.000,E1 87.020} C_DIS
LIN {X -0.069,Y -567.534,Z 865.274,A 0.000,B 0.000,C 90.000,E1 85.355} C_DIS
LIN {X 0.070,Y -567.753,Z 865.267,A 0.000,B 0.000,C 90.000,E1 83.970} C_DIS
LIN {X 0.155,Y -568.026,Z 865.259,A 0.000,B 0.000,C 90.000,E1 82.591} C_DIS
LIN {X 0.092,Y -568.616,Z 865.248,A 0.000,B 0.000,C 90.000,E1 80.679} C_DIS
LIN {X -0.042,Y -569.185,Z 865.239,A 0.000,B 0.000,C 90.000,E1 79.050} C_DIS
LIN {X 0.131,Y -570.015,Z 865.229,A 0.000,B 0.000,C 90.000,E1 77.117} C_DIS
LIN {X 0.082,Y -570.487,Z 865.221,A 0.000,B 0.000,C 90.000,E1 75.755} C_DIS
LIN {X 0.046,Y -570.900,Z 865.213,A 0.000,B 0.000,C 90.000,E1 74.393} C_DIS
LIN {X -0.171,Y -571.199,Z 865.207,A 0.000,B 0.000,C 90.000,E1 73.323} C_DIS
LIN {X 0.304,Y -571.424,Z 865.198,A 0.000,B 0.000,C 90.000,E1 71.638} C_DIS
LIN {X 0.236,Y -571.505,Z 865.189,A 0.000,B 0.000,C 90.000,E1 70.007} C_DIS
LIN {X -0.148,Y -571.544,Z 865.183,A 0.000,B 0.000,C 90.000,E1 68.954} C_DIS
LIN {X -0.165,Y -571.531,Z 865.175,A 0.000,B 0.000,C 90.000,E1 67.592} C_DIS
LIN {X -0.184,Y -571.538,Z 865.168,A 0.000,B 0.000,C 90.000,E1 66.230} C_DIS
LIN {X -0.144,Y -571.341,Z 865.159,A 0.000,B 0.000,C 90.000,E1 64.588} C_DIS
LIN {X 0.048,Y -571.017,Z 865.151,A 0.000,B 0.000,C 90.000,E1 63.204} C_DIS
LIN {X -0.026,Y -570.647,Z 865.144,A 0.000,B 0.000,C 90.000,E1 61.847} C_DIS
LIN {X 0.062,Y -570.209,Z 865.138,A 0.000,B 0.000,C 90.000,E1 60.745} C_DIS
LIN {X -0.071,Y -569.701,Z 865.131,A 0.000,B 0.000,C 90.000,E1 59.665} C_DIS
LIN {X 0.103,Y -568.685,Z 865.124,A 0.000,B 0.000,C 90.000,E1 58.280} C_DIS
LIN {X 0.146,Y -568.043,Z 865.119,A 0.000,B 0.000,C 90.000,E1 57.454} C_DIS
LIN {X 0.185,Y -567.245,Z 865.115,A 0.000,B 0.000,C 90.000,E1 56.628} C_DIS
LIN {X 0.014,Y -565.918,Z 865.109,A 0.000,B 0.000,C 90.000,E1 55.548} C_DIS
LIN {X 0.352,Y -564.810,Z 865.104,A 0.000,B 0.000,C 90.000,E1 54.689} C_DIS
LIN {X 0.003,Y -563.202,Z 865.098,A 0.000,B 0.000,C 90.000,E1 53.623} C_DIS
LIN {X -0.367,Y -561.329,Z 865.092,A 0.000,B 0.000,C 90.000,E1 52.557} C_DIS
LIN {X -0.076,Y -559.742,Z 865.087,A 0.000,B 0.000,C 90.000,E1 51.698} C_DIS
LIN {X -0.242,Y -557.949,Z 865.083,A 0.000,B 0.000,C 90.000,E1 50.884} C_DIS
LIN {X 0.280,Y -556.609,Z 865.080,A 0.000,B 0.000,C 90.000,E1 50.275} C_DIS
LIN {X 0.082,Y -554.280,Z 865.075,A 0.000,B 0.000,C 90.000,E1 49.461} C_DIS
LIN {X 0.221,Y -551.617,Z 865.070,A 0.000,B 0.000,C 90.000,E1 48.609} C_DIS
LIN {X -0.082,Y -549.733,Z 865.067,A 0.000,B 0.000,C 90.000,E1 48.081} C_DIS
LIN {X 0.010,Y -546.551,Z 865.062,A 0.000,B 0.000,C 90.000,E1 47.229} C_DIS
LIN {X -0.131,Y -543.652,Z 865.059,A 0.000,B 0.000,C 90.000,E1 46.539} C_DIS
LIN {X 0.071,Y -540.433,Z 865.055,A 0.000,B 0.000,C 90.000,E1 45.810} C_DIS
LIN {X 0.059,Y -537.644,Z 865.051,A 0.000,B 0.000,C 90.000,E1 45.243} C_DIS
LIN {X 0.028,Y -534.587,Z 865.048,A 0.000,B 0.000,C 90.000,E1 44.676} C_DIS
LIN {X 0.142,Y -530.330,Z 865.044,A 0.000,B 0.000,C 90.000,E1 43.947} C_DIS
LIN {X 0.055,Y -526.717,Z 865.041,A 0.000,B 0.000,C 90.000,E1 43.380} C_DIS
LIN {X -0.060,Y -522.849,Z 865.038,A 0.000,B 0.000,C 90.000,E1 42.813} C_DIS
LIN {X 0.037,Y -519.791,Z 865.035,A 0.000,B 0.000,C 90.000,E1 42.366} C_DIS
LIN {X 0.045,Y -514.249,Z 865.031,A 0.000,B 0.000,C 90.000,E1 41.634} C_DIS
LIN {X -0.285,Y -510.766,Z 865.029,A 0.000,B 0.000,C 90.000,E1 41.229} C_DIS
LIN {X -0.131,Y -505.735,Z 865.026,A 0.000,B 0.000,C 90.000,E1 40.620} C_DIS
LIN {X 0.064,Y -502.077,Z 865.023,A 0.000,B 0.000,C 90.000,E1 40.172} C_DIS
LIN {X -0.056,Y -498.251,Z 865.021,A 0.000,B 0.000,C 90.000,E1 39.769} C_DIS
LIN {X -0.060,Y -492.579,Z 865.018,A 0.000,B 0.000,C 90.000,E1 39.197} C_DIS
LIN {X 0.111,Y -484.262,Z 865.013,A 0.000,B 0.000,C 90.000,E1 38.382} C_DIS
LIN {X -0.218,Y -478.294,Z 865.010,A 0.000,B 0.000,C 90.000,E1 37.890} C_DIS
LIN {X 0.151,Y -469.234,Z 865.006,A 0.000,B 0.000,C 90.000,E1 37.076} C_DIS
LIN {X 0.101,Y -461.427,Z 865.003,A 0.000,B 0.000,C 90.000,E1 36.457} C_DIS
LIN {X 0.074,Y -452.093,Z 864.999,A 0.000,B 0.000,C 90.000,E1 35.724} C_DIS
LIN {X 0.177,Y -437.977,Z 864.992,A 0.000,B 0.000,C 90.000,E1 34.612} C_DIS
LIN {X 0.133,Y -419.366,Z 864.984,A 0.000,B 0.000,C 90.000,E1 33.086} C_DIS
LIN {X 0.108,Y -406.063,Z 864.977,A 0.000,B 0.000,C 90.000,E1 31.878} C_DIS
LIN {X -0.200,Y -400.329,Z 864.974,A 0.000,B 0.000,C 90.000,E1 31.337} C_DIS
LIN {X 0.046,Y -395.554,Z 864.971,A 0.000,B 0.000,C 90.000,E1 30.718} C_DIS
LIN {X -0.015,Y -393.071,Z 864.969,A 0.000,B 0.000,C 90.000,E1 30.335} C_DIS
LIN {X 0.046,Y -390.964,Z 864.966,A 0.000,B 0.000,C 90.000,E1 29.795} C_DIS
LIN {X -0.153,Y -390.049,Z 864.963,A 0.000,B 0.000,C 90.000,E1 29.283} C_DIS
LIN {X -0.019,Y -389.550,Z 864.958,A 0.000,B 0.000,C 90.000,E1 28.487} C_DIS
LIN {X 0.057,Y -390.220,Z 864.948,A 0.000,B 0.000,C 90.000,E1 26.693} C_DIS
LIN {X -0.101,Y -392.560,Z 864.931,A 0.000,B 0.000,C 90.000,E1 23.515} C_DIS
LIN {X 0.072,Y -395.558,Z 864.913,A 0.000,B 0.000,C 90.000,E1 20.301} C_DIS
LIN {X -0.061,Y -398.979,Z 864.895,A 0.000,B 0.000,C 90.000,E1 17.149} C_DIS
LIN {X -0.215,Y -402.065,Z 864.882,A 0.000,B 0.000,C 90.000,E1 14.717} C_DIS
LIN {X 0.116,Y -406.471,Z 864.864,A 0.000,B 0.000,C 90.000,E1 11.535} C_DIS
LIN {X -0.189,Y -409.699,Z 864.853,A 0.000,B 0.000,C 90.000,E1 9.500} C_DIS
LIN {X 0.007,Y -414.308,Z 864.837,A 0.000,B 0.000,C 90.000,E1 6.720} C_DIS
LIN {X 0.185,Y -418.043,Z 864.826,A 0.000,B 0.000,C 90.000,E1 4.645} C_DIS
LIN {X 0.102,Y -424.183,Z 864.809,A 0.000,B 0.000,C 90.000,E1 1.604} C_DIS
LIN {X -0.201,Y -429.113,Z 864.797,A 0.000,B 0.000,C 90.000,E1 359.484} C_DIS
LIN {X -0.170,Y -433.946,Z 864.786,A 0.000,B 0.000,C 90.000,E1 357.478} C_DIS
LIN {X -0.004,Y -438.959,Z 864.775,A 0.000,B 0.000,C 90.000,E1 355.469} C_DIS
LIN {X -0.203,Y -440.746,Z 864.771,A 0.000,B 0.000,C 90.000,E1 354.837} C_DIS
LIN {X 0.050,Y -442.864,Z 864.768,A 0.000,B 0.000,C 90.000,E1 354.147} C_DIS
LIN {X -0.155,Y -444.866,Z 864.765,A 0.000,B 0.000,C 90.000,E1 353.685} C_DIS
LIN {X 0.013,Y -446.761,Z 864.763,A 0.000,B 0.000,C 90.000,E1 353.337} C_DIS
LIN {X -0.157,Y -449.728,Z 864.761,A 0.000,B 0.000,C 90.000,E1 353.053} C_DIS
LIN {X 0.116,Y -451.252,Z 864.761,A 0.000,B 0.000,C 90.000,E1 352.875} C_DIS
LIN {X -0.003,Y -456.662,Z 864.759,A 0.000,B 0.000,C 90.000,E1 352.534} C_DIS
LIN {X -0.099,Y -469.338,Z 864.755,A 0.000,B 0.000,C 90.000,E1 351.951} C_DIS
LIN {X 0.092,Y -476.059,Z 864.753,A 0.000,B 0.000,C 90.000,E1 351.602} C_DIS
LIN {X 0.071,Y -485.835,Z 864.751,A 0.000,B 0.000,C 90.000,E1 351.084} C_DIS
LIN {X 0.151,Y -495.521,Z 864.747,A 0.000,B 0.000,C 90.000,E1 350.500} C_DIS
LIN {X 0.067,Y -506.512,Z 864.743,A 0.000,B 0.000,C 90.000,E1 349.803} C_DIS
LIN {X 0.078,Y -514.351,Z 864.741,A 0.000,B 0.000,C 90.000,E1 349.285} C_DIS
LIN {X -0.002,Y -522.088,Z 864.738,A 0.000,B 0.000,C 90.000,E1 348.757} C_DIS
LIN {X -0.216,Y -529.628,Z 864.735,A 0.000,B 0.000,C 90.000,E1 348.229} C_DIS
LIN {X -0.063,Y -535.509,Z 864.732,A 0.000,B 0.000,C 90.000,E1 347.757} C_DIS
LIN {X -0.188,Y -542.713,Z 864.729,A 0.000,B 0.000,C 90.000,E1 347.173} C_DIS
LIN {X 0.066,Y -551.044,Z 864.725,A 0.000,B 0.000,C 90.000,E1 346.408} C_DIS
LIN {X -0.056,Y -558.912,Z 864.720,A 0.000,B 0.000,C 90.000,E1 345.644} C_DIS
LIN {X -0.233,Y -565.193,Z 864.717,A 0.000,B 0.000,C 90.000,E1 344.991} C_DIS
LIN {X -0.120,Y -572.528,Z 864.712,A 0.000,B 0.000,C 90.000,E1 344.157} C_DIS
LIN {X 0.060,Y -579.005,Z 864.707,A 0.000,B 0.000,C 90.000,E1 343.323} C_DIS
LIN {X -0.249,Y -585.148,Z 864.703,A 0.000,B 0.000,C 90.000,E1 342.543} C_DIS
LIN {X -0.009,Y -591.531,Z 864.698,A 0.000,B 0.000,C 90.000,E1 341.583} C_DIS
LIN {X 0.051,Y -595.876,Z 864.694,A 0.000,B 0.000,C 90.000,E1 340.913} C_DIS
LIN {X -0.191,Y -602.105,Z 864.688,A 0.000,B 0.000,C 90.000,E1 339.880} C_DIS
LIN {X -0.138,Y -607.961,Z 864.682,A 0.000,B 0.000,C 90.000,E1 338.827} C_DIS
LIN {X 0.287,Y -615.706,Z 864.674,A 0.000,B 0.000,C 90.000,E1 337.358} C_DIS
LIN {X -0.043,Y -621.578,Z 864.668,A 0.000,B 0.000,C 90.000,E1 336.230} C_DIS
LIN {X -0.304,Y -625.131,Z 864.664,A 0.000,B 0.000,C 90.000,E1 335.485} C_DIS
LIN {X 0.314,Y -629.752,Z 864.658,A 0.000,B 0.000,C 90.000,E1 334.409} C_DIS
LIN {X -0.137,Y -633.936,Z 864.652,A 0.000,B 0.000,C 90.000,E1 333.435} C_DIS
LIN {X 0.040,Y -637.909,Z 864.647,A 0.000,B 0.000,C 90.000,E1 332.410} C_DIS
LIN {X 0.204,Y -640.662,Z 864.643,A 0.000,B 0.000,C 90.000,E1 331.641} C_DIS
LIN {X -0.036,Y -644.979,Z 864.636,A 0.000,B 0.000,C 90.000,E1 330.411} C_DIS
LIN {X 0.105,Y -649.116,Z 864.629,A 0.000,B 0.000,C 90.000,E1 329.154} C_DIS
LIN {X 0.100,Y -652.845,Z 864.622,A 0.000,B 0.000,C 90.000,E1 327.916} C_DIS
LIN {X 0.269,Y -655.549,Z 864.616,A 0.000,B 0.000,C 90.000,E1 326.914} C_DIS
LIN {X -0.181,Y -657.495,Z 864.612,A 0.000,B 0.000,C 90.000,E1 326.215} C_DIS
LIN {X -0.040,Y -660.370,Z 864.605,A 0.000,B 0.000,C 90.000,E1 324.975} C_DIS
LIN {X -0.008,Y -662.821,Z 864.599,A 0.000,B 0.000,C 90.000,E1 323.749} C_DIS
LIN {X 0.106,Y -664.531,Z 864.593,A 0.000,B 0.000,C 90.000,E1 322.763} C_DIS
LIN {X 0.210,Y -666.358,Z 864.586,A 0.000,B 0.000,C 90.000,E1 321.537} C_DIS
LIN {X -0.183,Y -668.002,Z 864.580,A 0.000,B 0.000,C 90.000,E1 320.356} C_DIS
LIN {X -0.118,Y -668.896,Z 864.576,A 0.000,B 0.000,C 90.000,E1 319.622} C_DIS
LIN {X -0.044,Y -670.236,Z 864.569,A 0.000,B 0.000,C 90.000,E1 318.405} C_DIS
LIN {X 0.092,Y -672.406,Z 864.558,A 0.000,B 0.000,C 90.000,E1 316.458} C_DIS
LIN {X 0.194,Y -673.961,Z 864.552,A 0.000,B 0.000,C 90.000,E1 315.243} C_DIS
LIN {X 0.218,Y -674.097,Z 864.550,A 0.000,B 0.000,C 90.000,E1 315.000} C_DIS
LIN {X 0.269,Y -674.670,Z 864.547,A 0.000,B 0.000,C 90.000,E1 314.514} C_DIS
LIN {X 0.059,Y -676.723,Z 864.535,A 0.000,B 0.000,C 90.000,E1 312.366} C_DIS
LIN {X 0.263,Y -677.891,Z 864.529,A 0.000,B 0.000,C 90.000,E1 311.148} C_DIS
LIN {X 0.079,Y -679.189,Z 864.521,A 0.000,B 0.000,C 90.000,E1 309.725} C_DIS
LIN {X -0.111,Y -680.208,Z 864.514,A 0.000,B 0.000,C 90.000,E1 308.543} C_DIS
LIN {X -0.118,Y -681.561,Z 864.505,A 0.000,B 0.000,C 90.000,E1 306.870} C_DIS
LIN {X -0.129,Y -682.643,Z 864.497,A 0.000,B 0.000,C 90.000,E1 305.438} C_DIS
LIN {X 0.043,Y -683.577,Z 864.489,A 0.000,B 0.000,C 90.000,E1 303.992} C_DIS
LIN {X 0.062,Y -684.903,Z 864.478,A 0.000,B 0.000,C 90.000,E1 302.084} C_DIS
LIN {X 0.131,Y -686.172,Z 864.469,A 0.000,B 0.000,C 90.000,E1 300.413} C_DIS
LIN {X 0.219,Y -687.560,Z 864.460,A 0.000,B 0.000,C 90.000,E1 298.743} C_DIS
LIN {X -0.183,Y -688.741,Z 864.453,A 0.000,B 0.000,C 90.000,E1 297.590} C_DIS
LIN {X -0.018,Y -690.185,Z 864.445,A 0.000,B 0.000,C 90.000,E1 296.155} C_DIS
LIN {X 0.241,Y -691.397,Z 864.439,A 0.000,B 0.000,C 90.000,E1 294.951} C_DIS
LIN {X -0.005,Y -692.168,Z 864.434,A 0.000,B 0.000,C 90.000,E1 294.027} C_DIS
LIN {X -0.196,Y -692.287,Z 864.430,A 0.000,B 0.000,C 90.000,E1 293.334} C_DIS
LIN {X 0.281,Y -691.528,Z 864.427,A 0.000,B 0.000,C 90.000,E1 292.823} C_DIS
LIN {X 0.250,Y -690.987,Z 864.426,A 0.000,B 0.000,C 90.000,E1 292.589} C_DIS
LIN {X -0.272,Y -690.456,Z 864.425,A 0.000,B 0.000,C 90.000,E1 292.514} C_DIS
LIN {X -0.188,Y -688.300,Z 864.423,A 0.000,B 0.000,C 90.000,E1 292.153} C_DIS
LIN {X 0.034,Y -686.450,Z 864.422,A 0.000,B 0.000,C 90.000,E1 291.897} C_DIS
LIN {X 0.141,Y -685.120,Z 864.421,A 0.000,B 0.000,C 90.000,E1 291.770} C_DIS
LIN {X -0.163,Y -681.377,Z 864.420,A 0.000,B 0.000,C 90.000,E1 291.589} C_DIS
LIN {X -0.255,Y -676.038,Z 864.419,A 0.000,B 0.000,C 90.000,E1 291.354} C_DIS
LIN {X -0.210,Y -669.633,Z 864.417,A 0.000,B 0.000,C 90.000,E1 291.153} C_DIS
LIN {X -0.131,Y -657.304,Z 864.416,A 0.000,B 0.000,C 90.000,E1 290.844} C_DIS
LIN {X -0.050,Y -655.580,Z 864.416,A 0.000,B 0.000,C 90.000,E1 290.791} C_DIS
LIN {X -0.080,Y -651.002,Z 864.414,A 0.000,B 0.000,C 90.000,E1 290.610} C_DIS
LIN {X -0.241,Y -649.682,Z 864.414,A 0.000,B 0.000,C 90.000,E1 290.556} C_DIS
LIN {X 0.155,Y -647.443,Z 864.413,A 0.000,B 0.000,C 90.000,E1 290.375} C_DIS
LIN {X 0.120,Y -647.419,Z 864.413,A 0.000,B 0.000,C 90.000,E1 290.375} C_DIS
LIN {X -0.204,Y -646.560,Z 864.412,A 0.000,B 0.000,C 90.000,E1 290.248} C_DIS
LIN {X -0.247,Y -646.549,Z 864.412,A 0.000,B 0.000,C 90.000,E1 290.248} C_DIS
LIN {X 0.304,Y -646.793,Z 864.411,A 0.000,B 0.000,C 90.000,E1 289.993} C_DIS
LIN {X 0.010,Y -648.284,Z 864.409,A 0.000,B 0.000,C 90.000,E1 289.631} C_DIS
LIN {X -0.140,Y -649.374,Z 864.408,A 0.000,B 0.000,C 90.000,E1 289.396} C_DIS
LIN {X -0.211,Y -655.372,Z 864.402,A 0.000,B 0.000,C 90.000,E1 288.290} C_DIS
LIN {X 0.329,Y -657.255,Z 864.400,A 0.000,B 0.000,C 90.000,E1 287.873} C_DIS
LIN {X 0.102,Y -659.626,Z 864.397,A 0.000,B 0.000,C 90.000,E1 287.402} C_DIS
LIN {X -0.016,Y -662.753,Z 864.393,A 0.000,B 0.000,C 90.000,E1 286.677} C_DIS
LIN {X -0.206,Y -664.587,Z 864.390,A 0.000,B 0.000,C 90.000,E1 286.205} C_DIS
LIN {X -0.285,Y -666.902,Z 864.386,A 0.000,B 0.000,C 90.000,E1 285.481} C_DIS
LIN {X 0.123,Y -668.746,Z 864.382,A 0.000,B 0.000,C 90.000,E1 284.717} C_DIS
LIN {X -0.022,Y -669.733,Z 864.379,A 0.000,B 0.000,C 90.000,E1 284.245} C_DIS
LIN {X -0.160,Y -670.550,Z 864.376,A 0.000,B 0.000,C 90.000,E1 283.772} C_DIS
LIN {X -0.359,Y -671.395,Z 864.372,A 0.000,B 0.000,C 90.000,E1 283.063} C_DIS
LIN {X 0.103,Y -671.999,Z 864.368,A 0.000,B 0.000,C 90.000,E1 282.299} C_DIS
LIN {X -0.025,Y -672.213,Z 864.366,A 0.000,B 0.000,C 90.000,E1 281.827} C_DIS
LIN {X -0.287,Y -672.230,Z 864.363,A 0.000,B 0.000,C 90.000,E1 281.366} C_DIS
LIN {X 0.244,Y -672.013,Z 864.360,A 0.000,B 0.000,C 90.000,E1 280.838} C_DIS
LIN {X 0.111,Y -671.572,Z 864.358,A 0.000,B 0.000,C 90.000,E1 280.366} C_DIS
LIN {X -0.147,Y -670.853,Z 864.355,A 0.000,B 0.000,C 90.000,E1 279.905} C_DIS
LIN {X 0.367,Y -669.873,Z 864.352,A 0.000,B 0.000,C 90.000,E1 279.378} C_DIS
LIN {X 0.182,Y -669.306,Z 864.351,A 0.000,B 0.000,C 90.000,E1 279.151} C_DIS
LIN {X 0.022,Y -667.908,Z 864.348,A 0.000,B 0.000,C 90.000,E1 278.681} C_DIS
LIN {X -0.251,Y -666.131,Z 864.346,A 0.000,B 0.000,C 90.000,E1 278.219} C_DIS
LIN {X 0.126,Y -664.027,Z 864.343,A 0.000,B 0.000,C 90.000,E1 277.701} C_DIS
LIN {X -0.276,Y -660.396,Z 864.339,A 0.000,B 0.000,C 90.000,E1 277.004} C_DIS
LIN {X 0.059,Y -657.489,Z 864.336,A 0.000,B 0.000,C 90.000,E1 276.486} C_DIS
LIN {X -0.279,Y -654.211,Z 864.333,A 0.000,B 0.000,C 90.000,E1 276.024} C_DIS
LIN {X -0.050,Y -650.349,Z 864.331,A 0.000,B 0.000,C 90.000,E1 275.511} C_DIS
LIN {X -0.317,Y -647.049,Z 864.329,A 0.000,B 0.000,C 90.000,E1 275.163} C_DIS
LIN {X 0.042,Y -643.498,Z 864.327,A 0.000,B 0.000,C 90.000,E1 274.759} C_DIS
LIN {X 0.070,Y -638.730,Z 864.324,A 0.000,B 0.000,C 90.000,E1 274.302} C_DIS
LIN {X 0.083,Y -631.827,Z 864.321,A 0.000,B 0.000,C 90.000,E1 273.726} C_DIS
LIN {X -0.140,Y -624.521,Z 864.318,A 0.000,B 0.000,C 90.000,E1 273.212} C_DIS
LIN {X 0.113,Y -616.706,Z 864.315,A 0.000,B 0.000,C 90.000,E1 272.694} C_DIS
LIN {X 0.017,Y -610.401,Z 864.313,A 0.000,B 0.000,C 90.000,E1 272.350} C_DIS
LIN {X 0.180,Y -603.692,Z 864.311,A 0.000,B 0.000,C 90.000,E1 272.007} C_DIS
LIN {X 0.160,Y -596.731,Z 864.310,A 0.000,B 0.000,C 90.000,E1 271.718} C_DIS
LIN {X -0.063,Y -591.287,Z 864.309,A 0.000,B 0.000,C 90.000,E1 271.547} C_DIS
LIN {X -0.013,Y -583.786,Z 864.307,A 0.000,B 0.000,C 90.000,E1 271.318} C_DIS
LIN {X -0.277,Y -577.665,Z 864.307,A 0.000,B 0.000,C 90.000,E1 271.203} C_DIS
LIN {X -0.119,Y -571.572,Z 864.306,A 0.000,B 0.000,C 90.000,E1 271.088} C_DIS
LIN {X -0.180,Y -565.780,Z 864.306,A 0.000,B 0.000,C 90.000,E1 271.031} C_DIS
LIN {X 0.272,Y -552.948,Z 864.305,A 0.000,B 0.000,C 90.000,E1 270.917} C_DIS
LIN {X 0.154,Y -550.373,Z 864.305,A 0.000,B 0.000,C 90.000,E1 270.859} C_DIS
LIN {X -0.059,Y -549.648,Z 864.305,A 0.000,B 0.000,C 90.000,E1 270.859} C_DIS
LIN {X -0.112,Y -549.555,Z 864.305,A 0.000,B 0.000,C 90.000,E1 270.859} C_DIS
LIN {X 0.176,Y -547.762,Z 864.304,A 0.000,B 0.000,C 90.000,E1 270.630} C_DIS
LIN {X 0.251,Y -546.761,Z 864.301,A 0.000,B 0.000,C 90.000,E1 270.229} C_DIS
LIN {X -0.249,Y -546.204,Z 864.300,A 0.000,B 0.000,C 90.000,E1 270.000} C_DIS
LIN {X -0.083,Y -544.950,Z 864.294,A 0.000,B 0.000,C 90.000,E1 268.854} C_DIS
LIN {X 0.227,Y -543.134,Z 864.281,A 0.000,B 0.000,C 90.000,E1 266.560} C_DIS
LIN {X -0.115,Y -542.232,Z 864.273,A 0.000,B 0.000,C 90.000,E1 265.179} C_DIS
LIN {X 0.065,Y -541.219,Z 864.265,A 0.000,B 0.000,C 90.000,E1 263.742} C_DIS
LIN {X 0.209,Y -540.315,Z 864.259,A 0.000,B 0.000,C 90.000,E1 262.591} C_DIS
LIN {X -0.058,Y -539.005,Z 864.251,A 0.000,B 0.000,C 90.000,E1 261.197} C_DIS
LIN {X 0.189,Y -537.659,Z 864.243,A 0.000,B 0.000,C 90.000,E1 259.746} C_DIS
LIN {X -0.081,Y -536.524,Z 864.237,A 0.000,B 0.000,C 90.000,E1 258.634} C_DIS
LIN {X 0.214,Y -534.964,Z 864.229,A 0.000,B 0.000,C 90.000,E1 257.173} C_DIS
LIN {X 0.075,Y -533.229,Z 864.221,A 0.000,B 0.000,C 90.000,E1 255.755} C_DIS
LIN {X 0.083,Y -531.115,Z 864.211,A 0.000,B 0.000,C 90.000,E1 254.031} C_DIS
LIN {X 0.036,Y -529.089,Z 864.202,A 0.000,B 0.000,C 90.000,E1 252.308} C_DIS
LIN {X 0.084,Y -527.325,Z 864.194,A 0.000,B 0.000,C 90.000,E1 250.859} C_DIS
LIN {X 0.275,Y -525.333,Z 864.186,A 0.000,B 0.000,C 90.000,E1 249.390} C_DIS
LIN {X -0.223,Y -523.782,Z 864.179,A 0.000,B 0.000,C 90.000,E1 248.284} C_DIS
LIN {X 0.099,Y -521.624,Z 864.171,A 0.000,B 0.000,C 90.000,E1 246.794} C_DIS
LIN {X -0.102,Y -519.367,Z 864.163,A 0.000,B 0.000,C 90.000,E1 245.357} C_DIS
LIN {X -0.126,Y -517.137,Z 864.155,A 0.000,B 0.000,C 90.000,E1 243.896} C_DIS
LIN {X 0.152,Y -514.116,Z 864.145,A 0.000,B 0.000,C 90.000,E1 242.103} C_DIS
LIN {X 0.146,Y -511.059,Z 864.135,A 0.000,B 0.000,C 90.000,E1 240.333} C_DIS
LIN {X 0.101,Y -508.865,Z 864.129,A 0.000,B 0.000,C 90.000,E1 239.154} C_DIS
LIN {X 0.172,Y -506.038,Z 864.120,A 0.000,B 0.000,C 90.000,E1 237.661} C_DIS
LIN {X -0.227,Y -503.122,Z 864.112,A 0.000,B 0.000,C 90.000,E1 236.215} C_DIS
LIN {X -0.154,Y -501.266,Z 864.107,A 0.000,B 0.000,C 90.000,E1 235.308} C_DIS
LIN {X 0.179,Y -498.475,Z 864.101,A 0.000,B 0.000,C 90.000,E1 234.069} C_DIS
LIN {X 0.217,Y -494.822,Z 864.092,A 0.000,B 0.000,C 90.000,E1 232.557} C_DIS
LIN {X 0.031,Y -490.489,Z 864.082,A 0.000,B 0.000,C 90.000,E1 230.759} C_DIS
LIN {X 0.162,Y -487.052,Z 864.074,A 0.000,B 0.000,C 90.000,E1 229.218} C_DIS
LIN {X 0.122,Y -480.882,Z 864.058,A 0.000,B 0.000,C 90.000,E1 226.458} C_DIS
LIN {X 0.291,Y -476.234,Z 864.046,A 0.000,B 0.000,C 90.000,E1 224.271} C_DIS
LIN {X -0.089,Y -472.124,Z 864.036,A 0.000,B 0.000,C 90.000,E1 222.447} C_DIS
LIN {X 0.060,Y -468.711,Z 864.027,A 0.000,B 0.000,C 90.000,E1 220.862} C_DIS
LIN {X 0.145,Y -465.335,Z 864.018,A 0.000,B 0.000,C 90.000,E1 219.277} C_DIS
LIN {X -0.133,Y -462.023,Z 864.010,A 0.000,B 0.000,C 90.000,E1 217.729} C_DIS
LIN {X -0.116,Y -458.720,Z 864.001,A 0.000,B 0.000,C 90.000,E1 216.137} C_DIS
LIN {X 0.037,Y -454.548,Z 863.990,A 0.000,B 0.000,C 90.000,E1 214.199} C_DIS
LIN {X 0.177,Y -449.780,Z 863.978,A 0.000,B 0.000,C 90.000,E1 211.926} C_DIS
LIN {X -0.047,Y -446.274,Z 863.969,A 0.000,B 0.000,C 90.000,E1 210.335} C_DIS
LIN {X 0.109,Y -442.227,Z 863.958,A 0.000,B 0.000,C 90.000,E1 208.359} C_DIS
LIN {X -0.050,Y -438.050,Z 863.947,A 0.000,B 0.000,C 90.000,E1 206.411} C_DIS
LIN {X 0.278,Y -433.921,Z 863.936,A 0.000,B 0.000,C 90.000,E1 204.387} C_DIS
LIN {X -0.234,Y -429.837,Z 863.925,A 0.000,B 0.000,C 90.000,E1 202.461} C_DIS
LIN {X 0.160,Y -426.433,Z 863.915,A 0.000,B 0.000,C 90.000,E1 200.737} C_DIS
LIN {X 0.120,Y -422.495,Z 863.904,A 0.000,B 0.000,C 90.000,E1 198.725} C_DIS
LIN {X 0.079,Y -419.219,Z 863.895,A 0.000,B 0.000,C 90.000,E1 197.040} C_DIS
LIN {X 0.054,Y -417.230,Z 863.889,A 0.000,B 0.000,C 90.000,E1 196.024} C_DIS
LIN {X 0.187,Y -413.727,Z 863.880,A 0.000,B 0.000,C 90.000,E1 194.300} C_DIS
LIN {X -0.095,Y -408.270,Z 863.864,A 0.000,B 0.000,C 90.000,E1 191.591} C_DIS
LIN {X -0.012,Y -404.919,Z 863.855,A 0.000,B 0.000,C 90.000,E1 189.849} C_DIS
LIN {X 0.009,Y -401.480,Z 863.845,A 0.000,B 0.000,C 90.000,E1 188.106} C_DIS
LIN {X 0.105,Y -395.475,Z 863.828,A 0.000,B 0.000,C 90.000,E1 184.935} C_DIS
LIN {X 0.135,Y -389.380,Z 863.806,A 0.000,B 0.000,C 90.000,E1 181.031} C_DIS
LIN {X 0.074,Y -386.918,Z 863.796,A 0.000,B 0.000,C 90.000,E1 179.255} C_DIS
LIN {X -0.030,Y -384.380,Z 863.786,A 0.000,B 0.000,C 90.000,E1 177.478} C_DIS
LIN {X -0.163,Y -381.824,Z 863.776,A 0.000,B 0.000,C 90.000,E1 175.698} C_DIS
LIN {X 0.101,Y -377.845,Z 863.760,A 0.000,B 0.000,C 90.000,E1 172.761} C_DIS
LIN {X 0.041,Y -373.697,Z 863.738,A 0.000,B 0.000,C 90.000,E1 168.757} C_DIS
LIN {X -0.160,Y -372.807,Z 863.725,A 0.000,B 0.000,C 90.000,E1 166.589} C_DIS
LIN {X 0.001,Y -372.736,Z 863.719,A 0.000,B 0.000,C 90.000,E1 165.463} C_DIS
LIN {X -0.165,Y -372.932,Z 863.715,A 0.000,B 0.000,C 90.000,E1 164.755} C_DIS
LIN {X 0.129,Y -373.530,Z 863.711,A 0.000,B 0.000,C 90.000,E1 163.976} C_DIS
LIN {X -0.048,Y -374.679,Z 863.706,A 0.000,B 0.000,C 90.000,E1 163.087} C_DIS
LIN {X -0.123,Y -376.084,Z 863.703,A 0.000,B 0.000,C 90.000,E1 162.489} C_DIS
LIN {X -0.133,Y -376.479,Z 863.702,A 0.000,B 0.000,C 90.000,E1 162.308} C_DIS
LIN {X -0.051,Y -378.713,Z 863.698,A 0.000,B 0.000,C 90.000,E1 161.692} C_DIS
LIN {X -0.122,Y -380.941,Z 863.696,A 0.000,B 0.000,C 90.000,E1 161.329} C_DIS
LIN {X -0.123,Y -383.027,Z 863.694,A 0.000,B 0.000,C 90.000,E1 160.967} C_DIS
LIN {X -0.121,Y -384.328,Z 863.693,A 0.000,B 0.000,C 90.000,E1 160.786} C_DIS
LIN {X -0.115,Y -385.927,Z 863.692,A 0.000,B 0.000,C 90.000,E1 160.604} C_DIS
LIN {X -0.067,Y -389.527,Z 863.691,A 0.000,B 0.000,C 90.000,E1 160.296} C_DIS
LIN {X -0.156,Y -391.101,Z 863.690,A 0.000,B 0.000,C 90.000,E1 160.188} C_DIS
LIN {X -0.125,Y -399.383,Z 863.687,A 0.000,B 0.000,C 90.000,E1 159.752} C_DIS
LIN {X -0.073,Y -406.303,Z 863.686,A 0.000,B 0.000,C 90.000,E1 159.444} C_DIS
LIN {X 0.171,Y -420.189,Z 863.682,A 0.000,B 0.000,C 90.000,E1 158.773} C_DIS
LIN {X -0.039,Y -423.250,Z 863.681,A 0.000,B 0.000,C 90.000,E1 158.646} C_DIS
LIN {X -0.108,Y -429.694,Z 863.679,A 0.000,B 0.000,C 90.000,E1 158.284} C_DIS
LIN {X 0.044,Y -437.621,Z 863.676,A 0.000,B 0.000,C 90.000,E1 157.741} C_DIS
LIN {X -0.070,Y -445.491,Z 863.673,A 0.000,B 0.000,C 90.000,E1 157.177} C_DIS
LIN {X 0.087,Y -452.974,Z 863.670,A 0.000,B 0.000,C 90.000,E1 156.561} C_DIS
LIN {X 0.122,Y -457.462,Z 863.668,A 0.000,B 0.000,C 90.000,E1 156.177} C_DIS
LIN {X 0.090,Y -466.182,Z 863.663,A 0.000,B 0.000,C 90.000,E1 155.357} C_DIS
LIN {X 0.015,Y -469.044,Z 863.662,A 0.000,B 0.000,C 90.000,E1 155.101} C_DIS
LIN {X 0.089,Y -478.217,Z 863.656,A 0.000,B 0.000,C 90.000,E1 154.101} C_DIS
LIN {X 0.018,Y -483.509,Z 863.653,A 0.000,B 0.000,C 90.000,E1 153.512} C_DIS
LIN {X 0.033,Y -489.624,Z 863.649,A 0.000,B 0.000,C 90.000,E1 152.743} C_DIS
LIN {X 0.015,Y -494.353,Z 863.645,A 0.000,B 0.000,C 90.000,E1 152.153} C_DIS
LIN {X 0.108,Y -496.512,Z 863.644,A 0.000,B 0.000,C 90.000,E1 151.897} C_DIS
LIN {X 0.015,Y -500.807,Z 863.641,A 0.000,B 0.000,C 90.000,E1 151.307} C_DIS
LIN {X 0.116,Y -504.314,Z 863.638,A 0.000,B 0.000,C 90.000,E1 150.845} C_DIS
LIN {X -0.136,Y -509.714,Z 863.634,A 0.000,B 0.000,C 90.000,E1 150.127} C_DIS
LIN {X -0.165,Y -513.826,Z 863.631,A 0.000,B 0.000,C 90.000,E1 149.537} C_DIS
LIN {X 0.166,Y -516.956,Z 863.628,A 0.000,B 0.000,C 90.000,E1 149.076} C_DIS
LIN {X 0.033,Y -527.038,Z 863.620,A 0.000,B 0.000,C 90.000,E1 147.502} C_DIS
LIN {X -0.001,Y -531.384,Z 863.616,A 0.000,B 0.000,C 90.000,E1 146.786} C_DIS
LIN {X -0.311,Y -537.863,Z 863.609,A 0.000,B 0.000,C 90.000,E1 145.674} C_DIS
LIN {X 0.169,Y -542.391,Z 863.604,A 0.000,B 0.000,C 90.000,E1 144.769} C_DIS
LIN {X 0.304,Y -548.377,Z 863.598,A 0.000,B 0.000,C 90.000,E1 143.623} C_DIS
LIN {X -0.022,Y -558.832,Z 863.587,A 0.000,B 0.000,C 90.000,E1 141.698} C_DIS
LIN {X -0.191,Y -566.896,Z 863.579,A 0.000,B 0.000,C 90.000,E1 140.194} C_DIS
LIN {X -0.276,Y -571.141,Z 863.574,A 0.000,B 0.000,C 90.000,E1 139.380} C_DIS
LIN {X -0.353,Y -577.138,Z 863.567,A 0.000,B 0.000,C 90.000,E1 138.162} C_DIS
LIN {X -0.224,Y -582.332,Z 863.561,A 0.000,B 0.000,C 90.000,E1 137.067} C_DIS
LIN {X 0.270,Y -588.397,Z 863.555,A 0.000,B 0.000,C 90.000,E1 135.810} C_DIS
LIN {X 0.214,Y -595.486,Z 863.547,A 0.000,B 0.000,C 90.000,E1 134.352} C_DIS
LIN {X -0.132,Y -602.152,Z 863.539,A 0.000,B 0.000,C 90.000,E1 132.933} C_DIS
LIN {X 0.157,Y -608.044,Z 863.531,A 0.000,B 0.000,C 90.000,E1 131.595} C_DIS
LIN {X 0.132,Y -613.540,Z 863.524,A 0.000,B 0.000,C 90.000,E1 130.297} C_DIS
LIN {X -0.029,Y -617.628,Z 863.518,A 0.000,B 0.000,C 90.000,E1 129.277} C_DIS
LIN {X -0.128,Y -621.585,Z 863.513,A 0.000,B 0.000,C 90.000,E1 128.257} C_DIS
LIN {X -0.022,Y -628.099,Z 863.503,A 0.000,B 0.000,C 90.000,E1 126.457} C_DIS
LIN {X 0.009,Y -631.644,Z 863.497,A 0.000,B 0.000,C 90.000,E1 125.438} C_DIS
LIN {X 0.234,Y -634.832,Z 863.491,A 0.000,B 0.000,C 90.000,E1 124.405} C_DIS
LIN {X 0.101,Y -636.394,Z 863.489,A 0.000,B 0.000,C 90.000,E1 123.913} C_DIS
LIN {X 0.046,Y -639.139,Z 863.483,A 0.000,B 0.000,C 90.000,E1 122.911} C_DIS
LIN {X 0.327,Y -641.035,Z 863.479,A 0.000,B 0.000,C 90.000,E1 122.133} C_DIS
LIN {X -0.085,Y -644.192,Z 863.470,A 0.000,B 0.000,C 90.000,E1 120.669} C_DIS
LIN {X -0.033,Y -645.946,Z 863.465,A 0.000,B 0.000,C 90.000,E1 119.667} C_DIS
LIN {X 0.044,Y -646.339,Z 863.463,A 0.000,B 0.000,C 90.000,E1 119.411} C_DIS
LIN {X 0.125,Y -646.596,Z 863.462,A 0.000,B 0.000,C 90.000,E1 119.155} C_DIS
LIN {X -0.277,Y -647.518,Z 863.459,A 0.000,B 0.000,C 90.000,E1 118.693} C_DIS
LIN {X 0.290,Y -648.694,Z 863.455,A 0.000,B 0.000,C 90.000,E1 117.897} C_DIS
LIN {X 0.173,Y -650.413,Z 863.448,A 0.000,B 0.000,C 90.000,E1 116.668} C_DIS
LIN {X 0.079,Y -651.062,Z 863.446,A 0.000,B 0.000,C 90.000,E1 116.181} C_DIS
LIN {X -0.207,Y -651.500,Z 863.441,A 0.000,B 0.000,C 90.000,E1 115.463} C_DIS
LIN {X -0.009,Y -651.964,Z 863.439,A 0.000,B 0.000,C 90.000,E1 114.951} C_DIS
LIN {X 0.022,Y -652.038,Z 863.435,A 0.000,B 0.000,C 90.000,E1 114.207} C_DIS
LIN {X 0.222,Y -651.940,Z 863.432,A 0.000,B 0.000,C 90.000,E1 113.695} C_DIS
LIN {X 0.061,Y -651.448,Z 863.430,A 0.000,B 0.000,C 90.000,E1 113.462} C_DIS
LIN {X 0.255,Y -649.834,Z 863.428,A 0.000,B 0.000,C 90.000,E1 112.950} C_DIS
LIN {X 0.182,Y -646.893,Z 863.425,A 0.000,B 0.000,C 90.000,E1 112.461} C_DIS
LIN {X 0.222,Y -645.896,Z 863.424,A 0.000,B 0.000,C 90.000,E1 112.333} C_DIS
LIN {X -0.143,Y -640.382,Z 863.422,A 0.000,B 0.000,C 90.000,E1 111.897} C_DIS
LIN {X 0.208,Y -636.724,Z 863.421,A 0.000,B 0.000,C 90.000,E1 111.663} C_DIS
LIN {X 0.023,Y -634.897,Z 863.420,A 0.000,B 0.000,C 90.000,E1 111.589} C_DIS
LIN {X 0.119,Y -633.625,Z 863.419,A 0.000,B 0.000,C 90.000,E1 111.482} C_DIS
LIN {X -0.255,Y -631.803,Z 863.419,A 0.000,B 0.000,C 90.000,E1 111.408} C_DIS
LIN {X -0.229,Y -627.797,Z 863.418,A 0.000,B 0.000,C 90.000,E1 111.227} C_DIS
LIN {X 0.015,Y -624.988,Z 863.417,A 0.000,B 0.000,C 90.000,E1 111.046} C_DIS
LIN {X -0.137,Y -595.973,Z 863.409,A 0.000,B 0.000,C 90.000,E1 109.685} C_DIS
LIN {X 0.195,Y -587.339,Z 863.407,A 0.000,B 0.000,C 90.000,E1 109.268} C_DIS
LIN {X -0.129,Y -580.085,Z 863.406,A 0.000,B 0.000,C 90.000,E1 109.033} C_DIS
LIN {X -0.136,Y -567.394,Z 863.404,A 0.000,B 0.000,C 90.000,E1 108.652} C_DIS
LIN {X -0.145,Y -565.985,Z 863.403,A 0.000,B 0.000,C 90.000,E1 108.598} C_DIS
LIN {X -0.026,Y -562.324,Z 863.402,A 0.000,B 0.000,C 90.000,E1 108.362} C_DIS
LIN {X -0.076,Y -561.045,Z 863.401,A 0.000,B 0.000,C 90.000,E1 108.181} C_DIS
LIN {X -0.163,Y -559.614,Z 863.398,A 0.000,B 0.000,C 90.000,E1 107.638} C_DIS
LIN {X -0.265,Y -559.181,Z 863.396,A 0.000,B 0.000,C 90.000,E1 107.221} C_DIS
LIN {X -0.213,Y -559.210,Z 863.386,A 0.000,B 0.000,C 90.000,E1 105.552} C_DIS
LIN {X -0.163,Y -559.769,Z 863.377,A 0.000,B 0.000,C 90.000,E1 103.883} C_DIS
LIN {X 0.178,Y -560.606,Z 863.368,A 0.000,B 0.000,C 90.000,E1 102.187} C_DIS
LIN {X 0.148,Y -561.904,Z 863.357,A 0.000,B 0.000,C 90.000,E1 100.254} C_DIS
LIN {X -0.278,Y -562.890,Z 863.349,A 0.000,B 0.000,C 90.000,E1 98.916} C_DIS
LIN {X -0.213,Y -563.848,Z 863.342,A 0.000,B 0.000,C 90.000,E1 97.530} C_DIS
LIN {X -0.127,Y -564.643,Z 863.334,A 0.000,B 0.000,C 90.000,E1 96.144} C_DIS
LIN {X 0.062,Y -565.420,Z 863.325,A 0.000,B 0.000,C 90.000,E1 94.473} C_DIS
LIN {X 0.108,Y -565.954,Z 863.317,A 0.000,B 0.000,C 90.000,E1 93.094} C_DIS
LIN {X 0.125,Y -566.344,Z 863.310,A 0.000,B 0.000,C 90.000,E1 91.718} C_DIS
LIN {X 0.139,Y -566.745,Z 863.302,A 0.000,B 0.000,C 90.000,E1 90.344} C_DIS
LIN {X -0.168,Y -567.194,Z 863.291,A 0.000,B 0.000,C 90.000,E1 88.453} C_DIS
LIN {X 0.136,Y -567.522,Z 863.281,A 0.000,B 0.000,C 90.000,E1 86.502} C_DIS
LIN {X -0.230,Y -567.783,Z 863.272,A 0.000,B 0.000,C 90.000,E1 84.894} C_DIS
LIN {X 0.026,Y -568.089,Z 863.262,A 0.000,B 0.000,C 90.000,E1 83.223} C_DIS
LIN {X 0.243,Y -568.769,Z 863.249,A 0.000,B 0.000,C 90.000,E1 80.735} C_DIS
LIN {X -0.260,Y -569.442,Z 863.238,A 0.000,B 0.000,C 90.000,E1 78.870} C_DIS
LIN {X -0.074,Y -570.253,Z 863.227,A 0.000,B 0.000,C 90.000,E1 76.937} C_DIS
LIN {X 0.113,Y -570.652,Z 863.221,A 0.000,B 0.000,C 90.000,E1 75.825} C_DIS
LIN {X 0.223,Y -571.042,Z 863.214,A 0.000,B 0.000,C 90.000,E1 74.448} C_DIS
LIN {X 0.188,Y -571.358,Z 863.206,A 0.000,B 0.000,C 90.000,E1 73.087} C_DIS
LIN {X 0.120,Y -571.573,Z 863.197,A 0.000,B 0.000,C 90.000,E1 71.456} C_DIS
LIN {X -0.128,Y -571.632,Z 863.186,A 0.000,B 0.000,C 90.000,E1 69.571} C_DIS
LIN {X -0.002,Y -571.637,Z 863.177,A 0.000,B 0.000,C 90.000,E1 67.922} C_DIS
LIN {X -0.199,Y -571.571,Z 863.168,A 0.000,B 0.000,C 90.000,E1 66.305} C_DIS
LIN {X -0.166,Y -571.396,Z 863.159,A 0.000,B 0.000,C 90.000,E1 64.665} C_DIS
LIN {X 0.111,Y -570.971,Z 863.150,A 0.000,B 0.000,C 90.000,E1 62.999} C_DIS
LIN {X 0.210,Y -570.686,Z 863.144,A 0.000,B 0.000,C 90.000,E1 61.897} C_DIS
LIN {X -0.195,Y -570.219,Z 863.138,A 0.000,B 0.000,C 90.000,E1 60.845} C_DIS
LIN {X -0.112,Y -569.712,Z 863.132,A 0.000,B 0.000,C 90.000,E1 59.744} C_DIS
LIN {X 0.356,Y -568.661,Z 863.124,A 0.000,B 0.000,C 90.000,E1 58.329} C_DIS
LIN {X 0.097,Y -568.013,Z 863.120,A 0.000,B 0.000,C 90.000,E1 57.533} C_DIS
LIN {X 0.250,Y -566.865,Z 863.114,A 0.000,B 0.000,C 90.000,E1 56.421} C_DIS
LIN {X 0.071,Y -565.496,Z 863.108,A 0.000,B 0.000,C 90.000,E1 55.341} C_DIS
LIN {X -0.273,Y -563.937,Z 863.101,A 0.000,B 0.000,C 90.000,E1 54.276} C_DIS
LIN {X 0.049,Y -562.652,Z 863.097,A 0.000,B 0.000,C 90.000,E1 53.417} C_DIS
LIN {X -0.089,Y -561.226,Z 863.092,A 0.000,B 0.000,C 90.000,E1 52.603} C_DIS
LIN {X 0.205,Y -559.622,Z 863.088,A 0.000,B 0.000,C 90.000,E1 51.743} C_DIS
LIN {X 0.042,Y -557.813,Z 863.083,A 0.000,B 0.000,C 90.000,E1 50.928} C_DIS
LIN {X -0.138,Y -555.685,Z 863.078,A 0.000,B 0.000,C 90.000,E1 50.114} C_DIS
LIN {X 0.010,Y -554.109,Z 863.075,A 0.000,B 0.000,C 90.000,E1 49.542} C_DIS
LIN {X 0.147,Y -551.449,Z 863.071,A 0.000,B 0.000,C 90.000,E1 48.690} C_DIS
LIN {X -0.110,Y -548.474,Z 863.066,A 0.000,B 0.000,C 90.000,E1 47.877} C_DIS
LIN {X -0.067,Y -546.330,Z 863.063,A 0.000,B 0.000,C 90.000,E1 47.310} C_DIS
LIN {X -0.210,Y -543.412,Z 863.059,A 0.000,B 0.000,C 90.000,E1 46.620} C_DIS
LIN {X -0.011,Y -540.169,Z 863.055,A 0.000,B 0.000,C 90.000,E1 45.891} C_DIS
LIN {X -0.025,Y -537.386,Z 863.052,A 0.000,B 0.000,C 90.000,E1 45.324} C_DIS
LIN {X -0.058,Y -534.313,Z 863.049,A 0.000,B 0.000,C 90.000,E1 44.757} C_DIS
LIN {X 0.056,Y -529.990,Z 863.045,A 0.000,B 0.000,C 90.000,E1 44.028} C_DIS
LIN {X -0.033,Y -526.370,Z 863.042,A 0.000,B 0.000,C 90.000,E1 43.461} C_DIS
LIN {X 0.234,Y -522.473,Z 863.038,A 0.000,B 0.000,C 90.000,E1 42.852} C_DIS
LIN {X 0.088,Y -518.270,Z 863.035,A 0.000,B 0.000,C 90.000,E1 42.285} C_DIS
LIN {X 0.085,Y -512.615,Z 863.031,A 0.000,B 0.000,C 90.000,E1 41.553} C_DIS
LIN {X -0.132,Y -507.759,Z 863.028,A 0.000,B 0.000,C 90.000,E1 40.987} C_DIS
LIN {X -0.174,Y -501.317,Z 863.024,A 0.000,B 0.000,C 90.000,E1 40.253} C_DIS
LIN {X -0.052,Y -497.281,Z 863.021,A 0.000,B 0.000,C 90.000,E1 39.806} C_DIS
LIN {X 0.300,Y -491.576,Z 863.018,A 0.000,B 0.000,C 90.000,E1 39.197} C_DIS
LIN {X 0.019,Y -482.978,Z 863.013,A 0.000,B 0.000,C 90.000,E1 38.418} C_DIS
LIN {X -0.095,Y -473.891,Z 863.009,A 0.000,B 0.000,C 90.000,E1 37.649} C_DIS
LIN {X 0.039,Y -466.286,Z 863.006,A 0.000,B 0.000,C 90.000,E1 36.996} C_DIS
LIN {X 0.074,Y -453.825,Z 863.000,A 0.000,B 0.000,C 90.000,E1 36.011} C_DIS
LIN {X 0.164,Y -439.630,Z 862.994,A 0.000,B 0.000,C 90.000,E1 34.898} C_DIS
LIN {X -0.117,Y -419.507,Z 862.985,A 0.000,B 0.000,C 90.000,E1 33.293} C_DIS
LIN {X 0.004,Y -406.076,Z 862.978,A 0.000,B 0.000,C 90.000,E1 32.054} C_DIS
LIN {X 0.027,Y -399.183,Z 862.974,A 0.000,B 0.000,C 90.000,E1 31.337} C_DIS
LIN {X -0.012,Y -395.304,Z 862.971,A 0.000,B 0.000,C 90.000,E1 30.846} C_DIS
LIN {X 0.027,Y -392.642,Z 862.969,A 0.000,B 0.000,C 90.000,E1 30.384} C_DIS
LIN {X -0.113,Y -390.820,Z 862.966,A 0.000,B 0.000,C 90.000,E1 29.873} C_DIS
LIN {X 0.008,Y -390.556,Z 862.964,A 0.000,B 0.000,C 90.000,E1 29.589} C_DIS
LIN {X 0.198,Y -390.005,Z 862.962,A 0.000,B 0.000,C 90.000,E1 29.205} C_DIS
LIN {X 0.235,Y -389.637,Z 862.958,A 0.000,B 0.000,C 90.000,E1 28.487} C_DIS
LIN {X -0.035,Y -390.355,Z 862.949,A 0.000,B 0.000,C 90.000,E1 26.744} C_DIS
LIN {X -0.036,Y -392.399,Z 862.933,A 0.000,B 0.000,C 90.000,E1 23.898} C_DIS
LIN {X 0.026,Y -394.602,Z 862.919,A 0.000,B 0.000,C 90.000,E1 21.408} C_DIS
LIN {X 0.162,Y -396.730,Z 862.907,A 0.000,B 0.000,C 90.000,E1 19.268} C_DIS
LIN {X 0.097,Y -399.079,Z 862.896,A 0.000,B 0.000,C 90.000,E1 17.166} C_DIS
LIN {X 0.150,Y -402.607,Z 862.880,A 0.000,B 0.000,C 90.000,E1 14.356} C_DIS
LIN {X 0.013,Y -407.100,Z 862.863,A 0.000,B 0.000,C 90.000,E1 11.243} C_DIS
LIN {X 0.153,Y -410.906,Z 862.849,A 0.000,B 0.000,C 90.000,E1 8.803} C_DIS
LIN {X -0.028,Y -416.276,Z 862.832,A 0.000,B 0.000,C 90.000,E1 5.739} C_DIS
LIN {X -0.179,Y -421.420,Z 862.817,A 0.000,B 0.000,C 90.000,E1 3.037} C_DIS
LIN {X -0.200,Y -429.272,Z 862.797,A 0.000,B 0.000,C 90.000,E1 359.484} C_DIS
LIN {X -0.081,Y -434.898,Z 862.784,A 0.000,B 0.000,C 90.000,E1 357.135} C_DIS
LIN {X -0.195,Y -440.865,Z 862.771,A 0.000,B 0.000,C 90.000,E1 354.837} C_DIS
LIN {X 0.059,Y -442.915,Z 862.768,A 0.000,B 0.000,C 90.000,E1 354.147} C_DIS
LIN {X -0.170,Y -444.796,Z 862.765,A 0.000,B 0.000,C 90.000,E1 353.685} C_DIS
LIN {X -0.003,Y -446.439,Z 862.763,A 0.000,B 0.000,C 90.000,E1 353.337} C_DIS
LIN {X -0.195,Y -446.957,Z 862.763,A 0.000,B 0.000,C 90.000,E1 353.280} C_DIS
LIN {X 0.144,Y -452.061,Z 862.760,A 0.000,B 0.000,C 90.000,E1 352.704} C_DIS
LIN {X 0.185,Y -457.407,Z 862.758,A 0.000,B 0.000,C 90.000,E1 352.356} C_DIS
LIN {X 0.154,Y -468.386,Z 862.755,A 0.000,B 0.000,C 90.000,E1 351.837} C_DIS
LIN {X 0.135,Y -473.536,Z 862.753,A 0.000,B 0.000,C 90.000,E1 351.602} C_DIS
LIN {X 0.198,Y -483.377,Z 862.751,A 0.000,B 0.000,C 90.000,E1 351.084} C_DIS
LIN {X 0.174,Y -496.150,Z 862.746,A 0.000,B 0.000,C 90.000,E1 350.330} C_DIS
LIN {X -0.046,Y -505.605,Z 862.743,A 0.000,B 0.000,C 90.000,E1 349.746} C_DIS
LIN {X 0.019,Y -513.501,Z 862.740,A 0.000,B 0.000,C 90.000,E1 349.218} C_DIS
LIN {X -0.107,Y -521.174,Z 862.737,A 0.000,B 0.000,C 90.000,E1 348.701} C_DIS
LIN {X 0.174,Y -528.797,Z 862.734,A 0.000,B 0.000,C 90.000,E1 348.117} C_DIS
LIN {X -0.157,Y -534.739,Z 862.732,A 0.000,B 0.000,C 90.000,E1 347.701} C_DIS
LIN {X -0.198,Y -541.828,Z 862.728,A 0.000,B 0.000,C 90.000,E1 347.117} C_DIS
LIN {X 0.026,Y -550.324,Z 862.724,A 0.000,B 0.000,C 90.000,E1 346.353} C_DIS
LIN {X -0.315,Y -555.542,Z 862.721,A 0.000,B 0.000,C 90.000,E1 345.880} C_DIS
LIN {X 0.139,Y -562.041,Z 862.718,A 0.000,B 0.000,C 90.000,E1 345.172} C_DIS
LIN {X 0.205,Y -570.709,Z 862.712,A 0.000,B 0.000,C 90.000,E1 344.212} C_DIS
LIN {X -0.159,Y -573.075,Z 862.711,A 0.000,B 0.000,C 90.000,E1 343.976} C_DIS
LIN {X -0.064,Y -580.558,Z 862.706,A 0.000,B 0.000,C 90.000,E1 343.015} C_DIS
LIN {X -0.278,Y -585.630,Z 862.702,A 0.000,B 0.000,C 90.000,E1 342.362} C_DIS
LIN {X -0.033,Y -592.016,Z 862.697,A 0.000,B 0.000,C 90.000,E1 341.402} C_DIS
LIN {X 0.032,Y -596.309,Z 862.693,A 0.000,B 0.000,C 90.000,E1 340.732} C_DIS
LIN {X -0.205,Y -602.545,Z 862.687,A 0.000,B 0.000,C 90.000,E1 339.699} C_DIS
LIN {X -0.146,Y -608.410,Z 862.681,A 0.000,B 0.000,C 90.000,E1 338.646} C_DIS
LIN {X -0.251,Y -614.764,Z 862.675,A 0.000,B 0.000,C 90.000,E1 337.486} C_DIS
LIN {X 0.246,Y -618.089,Z 862.671,A 0.000,B 0.000,C 90.000,E1 336.794} C_DIS
LIN {X -0.044,Y -621.959,Z 862.667,A 0.000,B 0.000,C 90.000,E1 336.049} C_DIS
LIN {X -0.033,Y -626.692,Z 862.661,A 0.000,B 0.000,C 90.000,E1 335.025} C_DIS
LIN {X -0.252,Y -630.150,Z 862.657,A 0.000,B 0.000,C 90.000,E1 334.280} C_DIS
LIN {X -0.133,Y -634.318,Z 862.651,A 0.000,B 0.000,C 90.000,E1 333.256} C_DIS
LIN {X 0.044,Y -638.282,Z 862.646,A 0.000,B 0.000,C 90.000,E1 332.231} C_DIS
LIN {X -0.357,Y -641.045,Z 862.642,A 0.000,B 0.000,C 90.000,E1 331.513} C_DIS
LIN {X 0.284,Y -645.396,Z 862.635,A 0.000,B 0.000,C 90.000,E1 330.205} C_DIS
LIN {X 0.356,Y -648.747,Z 862.629,A 0.000,B 0.000,C 90.000,E1 329.203} C_DIS
LIN {X 0.007,Y -652.522,Z 862.622,A 0.000,B 0.000,C 90.000,E1 327.995} C_DIS
LIN {X 0.076,Y -654.600,Z 862.618,A 0.000,B 0.000,C 90.000,E1 327.248} C_DIS
LIN {X -0.288,Y -657.259,Z 862.613,A 0.000,B 0.000,C 90.000,E1 326.294} C_DIS
LIN {X -0.154,Y -660.214,Z 862.606,A 0.000,B 0.000,C 90.000,E1 325.055} C_DIS
LIN {X -0.079,Y -662.257,Z 862.600,A 0.000,B 0.000,C 90.000,E1 324.069} C_DIS
LIN {X 0.019,Y -664.114,Z 862.595,A 0.000,B 0.000,C 90.000,E1 323.084} C_DIS
LIN {X 0.016,Y -665.676,Z 862.590,A 0.000,B 0.000,C 90.000,E1 322.110} C_DIS
LIN {X 0.135,Y -667.441,Z 862.583,A 0.000,B 0.000,C 90.000,E1 320.884} C_DIS
LIN {X 0.189,Y -668.726,Z 862.577,A 0.000,B 0.000,C 90.000,E1 319.908} C_DIS
LIN {X -0.173,Y -670.350,Z 862.569,A 0.000,B 0.000,C 90.000,E1 318.485} C_DIS
LIN {X -0.035,Y -672.566,Z 862.559,A 0.000,B 0.000,C 90.000,E1 316.539} C_DIS
LIN {X 0.068,Y -674.106,Z 862.552,A 0.000,B 0.000,C 90.000,E1 315.324} C_DIS
LIN {X 0.119,Y -674.519,Z 862.549,A 0.000,B 0.000,C 90.000,E1 314.838} C_DIS
LIN {X 0.145,Y -674.850,Z 862.548,A 0.000,B 0.000,C 90.000,E1 314.595} C_DIS
LIN {X -0.060,Y -676.894,Z 862.536,A 0.000,B 0.000,C 90.000,E1 312.447} C_DIS
LIN {X 0.148,Y -678.050,Z 862.529,A 0.000,B 0.000,C 90.000,E1 311.229} C_DIS
LIN {X -0.002,Y -679.587,Z 862.520,A 0.000,B 0.000,C 90.000,E1 309.564} C_DIS
LIN {X -0.217,Y -680.409,Z 862.515,A 0.000,B 0.000,C 90.000,E1 308.624} C_DIS
LIN {X -0.216,Y -681.763,Z 862.505,A 0.000,B 0.000,C 90.000,E1 306.950} C_DIS
LIN {X -0.220,Y -682.876,Z 862.497,A 0.000,B 0.000,C 90.000,E1 305.518} C_DIS
LIN {X -0.036,Y -683.955,Z 862.488,A 0.000,B 0.000,C 90.000,E1 303.833} C_DIS
LIN {X 0.357,Y -685.114,Z 862.479,A 0.000,B 0.000,C 90.000,E1 302.133} C_DIS
LIN {X 0.044,Y -686.555,Z 862.468,A 0.000,B 0.000,C 90.000,E1 300.256} C_DIS
LIN {X 0.173,Y -687.763,Z 862.460,A 0.000,B 0.000,C 90.000,E1 298.821} C_DIS
LIN {X 0.329,Y -689.137,Z 862.452,A 0.000,B 0.000,C 90.000,E1 297.385} C_DIS
LIN {X 0.192,Y -690.589,Z 862.444,A 0.000,B 0.000,C 90.000,E1 295.976} C_DIS
LIN {X -0.214,Y -692.000,Z 862.437,A 0.000,B 0.000,C 90.000,E1 294.591} C_DIS
LIN {X -0.125,Y -692.475,Z 862.433,A 0.000,B 0.000,C 90.000,E1 293.875} C_DIS
LIN {X 0.076,Y -692.487,Z 862.430,A 0.000,B 0.000,C 90.000,E1 293.387} C_DIS
LIN {X 0.042,Y -692.294,Z 862.429,A 0.000,B 0.000,C 90.000,E1 293.153} C_DIS
LIN {X -0.119,Y -691.320,Z 862.426,A 0.000,B 0.000,C 90.000,E1 292.695} C_DIS
LIN {X -0.151,Y -690.342,Z 862.425,A 0.000,B 0.000,C 90.000,E1 292.461} C_DIS
LIN {X 0.081,Y -688.775,Z 862.423,A 0.000,B 0.000,C 90.000,E1 292.206} C_DIS
LIN {X 0.048,Y -686.923,Z 862.422,A 0.000,B 0.000,C 90.000,E1 291.972} C_DIS
LIN {X 0.157,Y -685.873,Z 862.421,A 0.000,B 0.000,C 90.000,E1 291.844} C_DIS
LIN {X 0.265,Y -684.298,Z 862.421,A 0.000,B 0.000,C 90.000,E1 291.716} C_DIS
LIN {X -0.040,Y -680.149,Z 862.420,A 0.000,B 0.000,C 90.000,E1 291.535} C_DIS
LIN {X -0.319,Y -676.614,Z 862.419,A 0.000,B 0.000,C 90.000,E1 291.408} C_DIS
LIN {X -0.259,Y -671.377,Z 862.418,A 0.000,B 0.000,C 90.000,E1 291.227} C_DIS
LIN {X -0.085,Y -669.323,Z 862.418,A 0.000,B 0.000,C 90.000,E1 291.153} C_DIS
LIN {X -0.005,Y -656.631,Z 862.416,A 0.000,B 0.000,C 90.000,E1 290.844} C_DIS
LIN {X 0.057,Y -653.562,Z 862.415,A 0.000,B 0.000,C 90.000,E1 290.737} C_DIS
LIN {X 0.101,Y -650.450,Z 862.415,A 0.000,B 0.000,C 90.000,E1 290.610} C_DIS
LIN {X 0.030,Y -649.237,Z 862.414,A 0.000,B 0.000,C 90.000,E1 290.556} C_DIS
LIN {X 0.096,Y -646.241,Z 862.413,A 0.000,B 0.000,C 90.000,E1 290.355} C_DIS
LIN {X 0.062,Y -646.199,Z 862.413,A 0.000,B 0.000,C 90.000,E1 290.355} C_DIS
LIN {X 0.050,Y -645.602,Z 862.413,A 0.000,B 0.000,C 90.000,E1 290.248} C_DIS
LIN {X 0.005,Y -645.584,Z 862.413,A 0.000,B 0.000,C 90.000,E1 290.248} C_DIS
LIN {X -0.069,Y -645.964,Z 862.411,A 0.000,B 0.000,C 90.000,E1 289.939} C_DIS
LIN {X -0.195,Y -647.510,Z 862.409,A 0.000,B 0.000,C 90.000,E1 289.577} C_DIS
LIN {X -0.240,Y -650.019,Z 862.406,A 0.000,B 0.000,C 90.000,E1 289.087} C_DIS
LIN {X 0.251,Y -655.347,Z 862.400,A 0.000,B 0.000,C 90.000,E1 288.055} C_DIS
LIN {X 0.091,Y -658.833,Z 862.396,A 0.000,B 0.000,C 90.000,E1 287.330} C_DIS
LIN {X -0.128,Y -660.958,Z 862.394,A 0.000,B 0.000,C 90.000,E1 286.858} C_DIS
LIN {X -0.240,Y -663.777,Z 862.390,A 0.000,B 0.000,C 90.000,E1 286.134} C_DIS
LIN {X 0.132,Y -665.996,Z 862.385,A 0.000,B 0.000,C 90.000,E1 285.371} C_DIS
LIN {X -0.031,Y -667.292,Z 862.383,A 0.000,B 0.000,C 90.000,E1 284.898} C_DIS
LIN {X -0.096,Y -668.806,Z 862.379,A 0.000,B 0.000,C 90.000,E1 284.175} C_DIS
LIN {X -0.243,Y -669.603,Z 862.376,A 0.000,B 0.000,C 90.000,E1 283.703} C_DIS
LIN {X 0.195,Y -670.388,Z 862.372,A 0.000,B 0.000,C 90.000,E1 282.939} C_DIS
LIN {X -0.155,Y -670.978,Z 862.368,A 0.000,B 0.000,C 90.000,E1 282.243} C_DIS
LIN {X -0.221,Y -671.130,Z 862.367,A 0.000,B 0.000,C 90.000,E1 282.007} C_DIS
LIN {X 0.302,Y -671.188,Z 862.364,A 0.000,B 0.000,C 90.000,E1 281.478} C_DIS
LIN {X -0.031,Y -670.814,Z 862.360,A 0.000,B 0.000,C 90.000,E1 280.782} C_DIS
LIN {X -0.171,Y -670.344,Z 862.357,A 0.000,B 0.000,C 90.000,E1 280.310} C_DIS
LIN {X 0.226,Y -669.600,Z 862.355,A 0.000,B 0.000,C 90.000,E1 279.792} C_DIS
LIN {X 0.072,Y -668.554,Z 862.352,A 0.000,B 0.000,C 90.000,E1 279.321} C_DIS
LIN {X -0.198,Y -667.235,Z 862.349,A 0.000,B 0.000,C 90.000,E1 278.859} C_DIS
LIN {X -0.285,Y -666.477,Z 862.348,A 0.000,B 0.000,C 90.000,E1 278.624} C_DIS
LIN {X 0.094,Y -664.679,Z 862.345,A 0.000,B 0.000,C 90.000,E1 278.106} C_DIS
LIN {X -0.194,Y -662.477,Z 862.342,A 0.000,B 0.000,C 90.000,E1 277.644} C_DIS
LIN {X 0.144,Y -659.416,Z 862.339,A 0.000,B 0.000,C 90.000,E1 277.004} C_DIS
LIN {X -0.283,Y -655.648,Z 862.336,A 0.000,B 0.000,C 90.000,E1 276.429} C_DIS
LIN {X 0.019,Y -652.300,Z 862.333,A 0.000,B 0.000,C 90.000,E1 275.910} C_DIS
LIN {X 0.296,Y -648.305,Z 862.330,A 0.000,B 0.000,C 90.000,E1 275.391} C_DIS
LIN {X -0.156,Y -643.706,Z 862.327,A 0.000,B 0.000,C 90.000,E1 274.935} C_DIS
LIN {X 0.155,Y -637.319,Z 862.324,A 0.000,B 0.000,C 90.000,E1 274.302} C_DIS
LIN {X 0.221,Y -631.794,Z 862.321,A 0.000,B 0.000,C 90.000,E1 273.841} C_DIS
LIN {X 0.031,Y -624.539,Z 862.319,A 0.000,B 0.000,C 90.000,E1 273.326} C_DIS
LIN {X -0.207,Y -616.878,Z 862.316,A 0.000,B 0.000,C 90.000,E1 272.865} C_DIS
LIN {X 0.147,Y -610.387,Z 862.314,A 0.000,B 0.000,C 90.000,E1 272.465} C_DIS
LIN {X -0.306,Y -603.588,Z 862.312,A 0.000,B 0.000,C 90.000,E1 272.178} C_DIS
LIN {X -0.241,Y -598.446,Z 862.311,A 0.000,B 0.000,C 90.000,E1 271.949} C_DIS
LIN {X -0.026,Y -591.014,Z 862.309,A 0.000,B 0.000,C 90.000,E1 271.661} C_DIS
LIN {X -0.048,Y -585.244,Z 862.308,A 0.000,B 0.000,C 90.000,E1 271.489} C_DIS
LIN {X -0.222,Y -577.508,Z 862.307,A 0.000,B 0.000,C 90.000,E1 271.318} C_DIS
LIN {X -0.073,Y -570.955,Z 862.307,A 0.000,B 0.000,C 90.000,E1 271.203} C_DIS
LIN {X -0.027,Y -565.307,Z 862.306,A 0.000,B 0.000,C 90.000,E1 271.146} C_DIS
LIN {X 0.023,Y -554.488,Z 862.306,A 0.000,B 0.000,C 90.000,E1 271.088} C_DIS
LIN {X -0.114,Y -552.487,Z 862.306,A 0.000,B 0.000,C 90.000,E1 271.088} C_DIS
LIN {X -0.208,Y -550.110,Z 862.306,A 0.000,B 0.000,C 90.000,E1 271.031} C_DIS
LIN {X -0.239,Y -550.061,Z 862.306,A 0.000,B 0.000,C 90.000,E1 271.031} C_DIS
LIN {X -0.126,Y -547.548,Z 862.304,A 0.000,B 0.000,C 90.000,E1 270.745} C_DIS
LIN {X -0.166,Y -547.535,Z 862.304,A 0.000,B 0.000,C 90.000,E1 270.745} C_DIS
LIN {X 0.064,Y -546.286,Z 862.301,A 0.000,B 0.000,C 90.000,E1 270.115} C_DIS
LIN {X 0.004,Y -543.269,Z 862.282,A 0.000,B 0.000,C 90.000,E1 266.731} C_DIS
LIN {X 0.163,Y -542.370,Z 862.274,A 0.000,B 0.000,C 90.000,E1 265.298} C_DIS
LIN {X -0.137,Y -541.148,Z 862.265,A 0.000,B 0.000,C 90.000,E1 263.628} C_DIS
LIN {X 0.074,Y -540.196,Z 862.258,A 0.000,B 0.000,C 90.000,E1 262.470} C_DIS
LIN {X 0.197,Y -539.145,Z 862.252,A 0.000,B 0.000,C 90.000,E1 261.319} C_DIS
LIN {X -0.091,Y -537.846,Z 862.244,A 0.000,B 0.000,C 90.000,E1 259.926} C_DIS
LIN {X 0.222,Y -536.396,Z 862.236,A 0.000,B 0.000,C 90.000,E1 258.465} C_DIS
LIN {X -0.015,Y -534.844,Z 862.228,A 0.000,B 0.000,C 90.000,E1 257.061} C_DIS
LIN {X -0.160,Y -533.111,Z 862.220,A 0.000,B 0.000,C 90.000,E1 255.644} C_DIS
LIN {X 0.017,Y -530.655,Z 862.209,A 0.000,B 0.000,C 90.000,E1 253.614} C_DIS
LIN {X 0.120,Y -528.640,Z 862.199,A 0.000,B 0.000,C 90.000,E1 251.873} C_DIS
LIN {X -0.009,Y -527.195,Z 862.193,A 0.000,B 0.000,C 90.000,E1 250.732} C_DIS
LIN {X -0.158,Y -524.462,Z 862.182,A 0.000,B 0.000,C 90.000,E1 248.720} C_DIS
LIN {X 0.173,Y -522.343,Z 862.174,A 0.000,B 0.000,C 90.000,E1 247.230} C_DIS
LIN {X -0.012,Y -520.152,Z 862.166,A 0.000,B 0.000,C 90.000,E1 245.793} C_DIS
LIN {X -0.220,Y -517.000,Z 862.154,A 0.000,B 0.000,C 90.000,E1 243.768} C_DIS
LIN {X 0.054,Y -513.898,Z 862.144,A 0.000,B 0.000,C 90.000,E1 241.975} C_DIS
LIN {X 0.044,Y -510.881,Z 862.135,A 0.000,B 0.000,C 90.000,E1 240.205} C_DIS
LIN {X 0.219,Y -507.528,Z 862.125,A 0.000,B 0.000,C 90.000,E1 238.408} C_DIS
LIN {X -0.156,Y -504.612,Z 862.116,A 0.000,B 0.000,C 90.000,E1 236.962} C_DIS
LIN {X -0.347,Y -502.836,Z 862.111,A 0.000,B 0.000,C 90.000,E1 236.087} C_DIS
LIN {X -0.278,Y -500.942,Z 862.106,A 0.000,B 0.000,C 90.000,E1 235.182} C_DIS
LIN {X 0.340,Y -498.133,Z 862.100,A 0.000,B 0.000,C 90.000,E1 233.909} C_DIS
LIN {X 0.094,Y -493.063,Z 862.088,A 0.000,B 0.000,C 90.000,E1 231.823} C_DIS
LIN {X 0.164,Y -487.438,Z 862.074,A 0.000,B 0.000,C 90.000,E1 229.380} C_DIS
LIN {X 0.134,Y -481.242,Z 862.059,A 0.000,B 0.000,C 90.000,E1 226.620} C_DIS
LIN {X 0.198,Y -477.207,Z 862.049,A 0.000,B 0.000,C 90.000,E1 224.757} C_DIS
LIN {X 0.067,Y -473.892,Z 862.040,A 0.000,B 0.000,C 90.000,E1 223.218} C_DIS
LIN {X -0.107,Y -470.439,Z 862.031,A 0.000,B 0.000,C 90.000,E1 221.676} C_DIS
LIN {X -0.058,Y -467.732,Z 862.025,A 0.000,B 0.000,C 90.000,E1 220.415} C_DIS
LIN {X 0.008,Y -464.399,Z 862.016,A 0.000,B 0.000,C 90.000,E1 218.830} C_DIS
LIN {X -0.038,Y -461.749,Z 862.009,A 0.000,B 0.000,C 90.000,E1 217.569} C_DIS
LIN {X 0.069,Y -458.432,Z 862.000,A 0.000,B 0.000,C 90.000,E1 215.964} C_DIS
LIN {X 0.204,Y -453.583,Z 861.987,A 0.000,B 0.000,C 90.000,E1 213.706} C_DIS
LIN {X -0.095,Y -450.198,Z 861.979,A 0.000,B 0.000,C 90.000,E1 212.133} C_DIS
LIN {X -0.081,Y -446.648,Z 861.969,A 0.000,B 0.000,C 90.000,E1 210.512} C_DIS
LIN {X -0.137,Y -442.622,Z 861.959,A 0.000,B 0.000,C 90.000,E1 208.565} C_DIS
LIN {X 0.114,Y -438.513,Z 861.948,A 0.000,B 0.000,C 90.000,E1 206.565} C_DIS
LIN {X 0.077,Y -433.712,Z 861.935,A 0.000,B 0.000,C 90.000,E1 204.259} C_DIS
LIN {X 0.142,Y -430.286,Z 861.926,A 0.000,B 0.000,C 90.000,E1 202.589} C_DIS
LIN {X 0.147,Y -426.908,Z 861.916,A 0.000,B 0.000,C 90.000,E1 200.918} C_DIS
LIN {X -0.071,Y -423.639,Z 861.907,A 0.000,B 0.000,C 90.000,E1 199.268} C_DIS
